LIN {X 0,Y 476.078,Z 721.43,A -85,B 0,C 180,E1 21900.686,E2 21900.686} C_VEL
LIN {X 0,Y 474.014,Z 739.797,A -85,B 0,C 180,E1 21899.021,E2 21899.021} C_VEL
LIN {X 0,Y 472.024,Z 756.489,A -85,B 0,C 180,E1 21897.228,E2 21897.228} C_VEL
LIN {X 0,Y 470.405,Z 770.596,A -85,B 0,C 180,E1 21895.493,E2 21895.493} C_VEL
LIN {X 0,Y 468.622,Z 786.231,A -85,B 0,C 180,E1 21893.248,E2 21893.248} C_VEL
LIN {X 0,Y 467.305,Z 798.417,A -85,B 0,C 180,E1 21891.198,E2 21891.198} C_VEL
LIN {X 0,Y 466.282,Z 809.049,A -85,B 0,C 180,E1 21889.152,E2 21889.152} C_VEL
LIN {X 0,Y 465.286,Z 820.849,A -85,B 0,C 180,E1 21886.478,E2 21886.478} C_VEL
LIN {X 0,Y 464.694,Z 829.202,A -85,B 0,C 180,E1 21884.198,E2 21884.198} C_VEL
LIN {X 0,Y 464.302,Z 836.544,A -85,B 0,C 180,E1 21881.805,E2 21881.805} C_VEL
LIN {X 0,Y 464.048,Z 843.148,A -85,B 0,C 180,E1 21879.049,E2 21879.049} C_VEL
LIN {X 0,Y 463.95,Z 847.377,A -85,B 0,C 180,E1 21876.683,E2 21876.683} C_VEL
LIN {X 0,Y 463.916,Z 850.478,A -85,B 0,C 180,E1 21874.202,E2 21874.202} C_VEL
LIN {X 0,Y 463.901,Z 852.199,A -85,B 0,C 180,E1 21871.482,E2 21871.482} C_VEL
LIN {X 0,Y 463.906,Z 852.333,A -85,B 0,C 180,E1 21869.136,E2 21869.136} C_VEL
LIN {X 0,Y 463.915,Z 851.272,A -85,B 0,C 180,E1 21866.788,E2 21866.788} C_VEL
LIN {X 0,Y 463.938,Z 848.514,A -85,B 0,C 180,E1 21864.062,E2 21864.062} C_VEL
LIN {X 0,Y 464.017,Z 844.133,A -85,B 0,C 180,E1 21861.45,E2 21861.45} C_VEL
LIN {X 0,Y 464.188,Z 839.084,A -85,B 0,C 180,E1 21859.179,E2 21859.179} C_VEL
LIN {X 0,Y 464.572,Z 831.33,A -85,B 0,C 180,E1 21856.433,E2 21856.433} C_VEL
LIN {X 0,Y 465.126,Z 822.811,A -85,B 0,C 180,E1 21854.029,E2 21854.029} C_VEL
LIN {X 0,Y 465.9,Z 813.253,A -85,B 0,C 180,E1 21851.741,E2 21851.741} C_VEL
LIN {X 0,Y 467.095,Z 800.545,A -85,B 0,C 180,E1 21849.186,E2 21849.186} C_VEL
LIN {X 0,Y 468.267,Z 789.404,A -85,B 0,C 180,E1 21847.265,E2 21847.265} C_VEL
LIN {X 0,Y 469.696,Z 776.705,A -85,B 0,C 180,E1 21845.341,E2 21845.341} C_VEL
LIN {X 0,Y 471.648,Z 759.814,A -85,B 0,C 180,E1 21843.158,E2 21843.158} C_VEL
LIN {X 0,Y 473.329,Z 745.351,A -85,B 0,C 180,E1 21841.554,E2 21841.554} C_VEL
LIN {X 0,Y 475.189,Z 729.447,A -85,B 0,C 180,E1 21840.009,E2 21840.009} C_VEL
LIN {X 0,Y 477.4,Z 709.425,A -85,B 0,C 180,E1 21838.357,E2 21838.357} C_VEL
LIN {X 0,Y 479.116,Z 692.979,A -85,B 0,C 180,E1 21837.212,E2 21837.212} C_VEL
LIN {X 0,Y 480.757,Z 675.933,A -85,B 0,C 180,E1 21836.198,E2 21836.198} C_VEL
LIN {X 0,Y 482.578,Z 654.654,A -85,B 0,C 180,E1 21835.158,E2 21835.158} C_VEL
LIN {X 0,Y 483.957,Z 634.596,A -85,B 0,C 180,E1 21834.403,E2 21834.403} C_VEL
LIN {X 0,Y 485.007,Z 616.285,A -85,B 0,C 180,E1 21833.877,E2 21833.877} C_VEL
LIN {X 0,Y 485.886,Z 591.815,A -85,B 0,C 180,E1 21833.389,E2 21833.389} C_VEL
LIN {X 0,Y 490.39,Z 370.649,A -85,B 0,C 180,E1 21829.748,E2 21829.748} C_VEL
LIN {X 0,Y 490.854,Z 340.827,A -85,B 0,C 180,E1 21829.233,E2 21829.233} C_VEL
LIN {X 0,Y 487.266,Z 328.463,A -85,B 0,C 180,E1 21828.634,E2 21828.634} C_VEL
LIN {X 0,Y 474.742,Z 306.974,A -85,B 0,C 180,E1 21826.867,E2 21826.867} C_VEL
LIN {X 0,Y 471.808,Z 301.758,A -85,B 0,C 180,E1 21826.372,E2 21826.372} C_VEL
LIN {X 0,Y 467.061,Z 288.332,A -85,B 0,C 180,E1 21823.746,E2 21823.746} C_VEL
LIN {X 0,Y 464.967,Z 282.439,A -85,B 0,C 180,E1 21822.471,E2 21822.471} C_VEL
LIN {X 0,Y 464.991,Z 282.262,A -85,B 0,C 180,E1 21819.052,E2 21819.052} C_VEL
LIN {X 0,Y 464.994,Z 282.317,A -85,B 0,C 180,E1 21815.42,E2 21815.42} C_VEL
LIN {X 0,Y 464.961,Z 282.319,A -85,B 0,C 180,E1 21811.855,E2 21811.855} C_VEL
LIN {X 0,Y 464.957,Z 282.317,A -85,B 0,C 180,E1 21808.235,E2 21808.235} C_VEL
LIN {X 0,Y 464.982,Z 282.302,A -85,B 0,C 180,E1 21804.655,E2 21804.655} C_VEL
LIN {X 0,Y 465.012,Z 282.287,A -85,B 0,C 180,E1 21801.068,E2 21801.068} C_VEL
LIN {X 0,Y 464.975,Z 282.314,A -85,B 0,C 180,E1 21797.521,E2 21797.521} C_VEL
LIN {X 0,Y 464.96,Z 282.299,A -85,B 0,C 180,E1 21793.936,E2 21793.936} C_VEL
LIN {X 0,Y 464.984,Z 282.3,A -85,B 0,C 180,E1 21790.406,E2 21790.406} C_VEL
LIN {X 0,Y 465.019,Z 282.307,A -85,B 0,C 180,E1 21786.792,E2 21786.792} C_VEL
LIN {X 0,Y 464.995,Z 282.287,A -85,B 0,C 180,E1 21783.081,E2 21783.081} C_VEL
LIN {X 0,Y 464.972,Z 282.315,A -85,B 0,C 180,E1 21779.507,E2 21779.507} C_VEL
LIN {X 0,Y 464.971,Z 282.294,A -85,B 0,C 180,E1 21775.807,E2 21775.807} C_VEL
LIN {X 0,Y 464.998,Z 282.304,A -85,B 0,C 180,E1 21772.215,E2 21772.215} C_VEL
LIN {X 0,Y 465.014,Z 282.303,A -85,B 0,C 180,E1 21768.591,E2 21768.591} C_VEL
LIN {X 0,Y 464.998,Z 282.289,A -85,B 0,C 180,E1 21764.919,E2 21764.919} C_VEL
LIN {X 0,Y 464.98,Z 282.315,A -85,B 0,C 180,E1 21761.313,E2 21761.313} C_VEL
LIN {X 0,Y 464.983,Z 282.313,A -85,B 0,C 180,E1 21757.609,E2 21757.609} C_VEL
LIN {X 0,Y 465.005,Z 282.311,A -85,B 0,C 180,E1 21753.983,E2 21753.983} C_VEL
LIN {X 0,Y 465.019,Z 282.311,A -85,B 0,C 180,E1 21750.3,E2 21750.3} C_VEL
LIN {X 0,Y 465.01,Z 282.311,A -85,B 0,C 180,E1 21746.602,E2 21746.602} C_VEL
LIN {X 0,Y 464.993,Z 282.314,A -85,B 0,C 180,E1 21742.913,E2 21742.913} C_VEL
LIN {X 0,Y 464.99,Z 282.313,A -85,B 0,C 180,E1 21739.343,E2 21739.343} C_VEL
LIN {X 0,Y 465.007,Z 282.311,A -85,B 0,C 180,E1 21735.668,E2 21735.668} C_VEL
LIN {X 0,Y 465.015,Z 282.312,A -85,B 0,C 180,E1 21731.931,E2 21731.931} C_VEL
LIN {X 0,Y 465.018,Z 282.312,A -85,B 0,C 180,E1 21728.26,E2 21728.26} C_VEL
LIN {X 0,Y 465.002,Z 282.312,A -85,B 0,C 180,E1 21724.56,E2 21724.56} C_VEL
LIN {X 0,Y 464.994,Z 282.311,A -85,B 0,C 180,E1 21720.913,E2 21720.913} C_VEL
LIN {X 0,Y 465.005,Z 282.307,A -85,B 0,C 180,E1 21717.257,E2 21717.257} C_VEL
LIN {X 0,Y 465.013,Z 282.308,A -85,B 0,C 180,E1 21713.573,E2 21713.573} C_VEL
LIN {X 0,Y 465.01,Z 282.31,A -85,B 0,C 180,E1 21709.86,E2 21709.86} C_VEL
LIN {X 0,Y 465.011,Z 282.31,A -85,B 0,C 180,E1 21709.539,E2 21709.539} C_VEL
LIN {X 0,Y 464.032,Z 282.435,A -85,B 0,C 180,E1 21708.59,E2 21708.59} C_VEL
LIN {X 0,Y 457.52,Z 283.245,A -85,B 0,C 180,E1 21705.85,E2 21705.85} C_VEL
LIN {X 0,Y 457.076,Z 283.3,A -85,B 0,C 180,E1 21705.223,E2 21705.223} C_VEL
LIN {X 0,Y 457.07,Z 283.302,A -85,B 0,C 180,E1 21701.474,E2 21701.474} C_VEL
LIN {X 0,Y 457.067,Z 283.304,A -85,B 0,C 180,E1 21697.71,E2 21697.71} C_VEL
LIN {X 0,Y 457.069,Z 283.302,A -85,B 0,C 180,E1 21694.014,E2 21694.014} C_VEL
LIN {X 0,Y 457.069,Z 283.301,A -85,B 0,C 180,E1 21690.251,E2 21690.251} C_VEL
LIN {X 0,Y 457.065,Z 283.301,A -85,B 0,C 180,E1 21686.488,E2 21686.488} C_VEL
LIN {X 0,Y 457.072,Z 283.3,A -85,B 0,C 180,E1 21682.711,E2 21682.711} C_VEL
LIN {X 0,Y 457.067,Z 283.301,A -85,B 0,C 180,E1 21679.029,E2 21679.029} C_VEL
LIN {X 0,Y 457.059,Z 283.304,A -85,B 0,C 180,E1 21675.3,E2 21675.3} C_VEL
LIN {X 0,Y 457.068,Z 283.302,A -85,B 0,C 180,E1 21671.639,E2 21671.639} C_VEL
LIN {X 0,Y 457.078,Z 283.299,A -85,B 0,C 180,E1 21667.899,E2 21667.899} C_VEL
LIN {X 0,Y 457.073,Z 283.298,A -85,B 0,C 180,E1 21664.195,E2 21664.195} C_VEL
LIN {X 0,Y 457.077,Z 283.297,A -85,B 0,C 180,E1 21660.516,E2 21660.516} C_VEL
LIN {X 0,Y 457.059,Z 283.3,A -85,B 0,C 180,E1 21656.847,E2 21656.847} C_VEL
LIN {X 0,Y 457.056,Z 283.301,A -85,B 0,C 180,E1 21653.174,E2 21653.174} C_VEL
LIN {X 0,Y 457.07,Z 283.3,A -85,B 0,C 180,E1 21649.483,E2 21649.483} C_VEL
LIN {X 0,Y 457.074,Z 283.3,A -85,B 0,C 180,E1 21645.749,E2 21645.749} C_VEL
LIN {X 0,Y 457.075,Z 283.301,A -85,B 0,C 180,E1 21642.019,E2 21642.019} C_VEL
LIN {X 0,Y 457.058,Z 283.301,A -85,B 0,C 180,E1 21638.409,E2 21638.409} C_VEL
LIN {X 0,Y 457.047,Z 283.304,A -85,B 0,C 180,E1 21634.818,E2 21634.818} C_VEL
LIN {X 0,Y 457.056,Z 283.303,A -85,B 0,C 180,E1 21631.083,E2 21631.083} C_VEL
LIN {X 0,Y 457.076,Z 283.302,A -85,B 0,C 180,E1 21627.488,E2 21627.488} C_VEL
LIN {X 0,Y 457.077,Z 283.3,A -85,B 0,C 180,E1 21623.735,E2 21623.735} C_VEL
LIN {X 0,Y 457.056,Z 283.3,A -85,B 0,C 180,E1 21620.087,E2 21620.087} C_VEL
LIN {X 0,Y 457.035,Z 283.286,A -85,B 0,C 180,E1 21616.523,E2 21616.523} C_VEL
LIN {X 0,Y 457.05,Z 283.305,A -85,B 0,C 180,E1 21612.893,E2 21612.893} C_VEL
LIN {X 0,Y 457.069,Z 283.273,A -85,B 0,C 180,E1 21609.189,E2 21609.189} C_VEL
LIN {X 0,Y 457.073,Z 283.296,A -85,B 0,C 180,E1 21605.523,E2 21605.523} C_VEL
LIN {X 0,Y 457.043,Z 283.292,A -85,B 0,C 180,E1 21601.88,E2 21601.88} C_VEL
LIN {X 0,Y 457.028,Z 283.286,A -85,B 0,C 180,E1 21598.245,E2 21598.245} C_VEL
LIN {X 0,Y 457.039,Z 283.305,A -85,B 0,C 180,E1 21594.602,E2 21594.602} C_VEL
LIN {X 0,Y 457.07,Z 283.272,A -85,B 0,C 180,E1 21591.065,E2 21591.065} C_VEL
LIN {X 0,Y 457.065,Z 283.301,A -85,B 0,C 180,E1 21587.324,E2 21587.324} C_VEL
LIN {X 0,Y 457.031,Z 283.294,A -85,B 0,C 180,E1 21583.738,E2 21583.738} C_VEL
LIN {X 0,Y 457.019,Z 283.283,A -85,B 0,C 180,E1 21580.044,E2 21580.044} C_VEL
LIN {X 0,Y 457.033,Z 283.303,A -85,B 0,C 180,E1 21576.4,E2 21576.4} C_VEL
LIN {X 0,Y 457.066,Z 283.291,A -85,B 0,C 180,E1 21572.794,E2 21572.794} C_VEL
LIN {X 0,Y 457.044,Z 283.29,A -85,B 0,C 180,E1 21569.209,E2 21569.209} C_VEL
LIN {X 0,Y 457.015,Z 283.297,A -85,B 0,C 180,E1 21565.636,E2 21565.636} C_VEL
LIN {X 0,Y 457.008,Z 283.254,A -85,B 0,C 180,E1 21561.905,E2 21561.905} C_VEL
LIN {X 0,Y 457.06,Z 283.456,A -85,B 0,C 180,E1 21558.358,E2 21558.358} C_VEL
LIN {X 0,Y 461.683,Z 296.244,A -85,B 0,C 180,E1 21555.612,E2 21555.612} C_VEL
LIN {X 0,Y 463.685,Z 301.866,A -85,B 0,C 180,E1 21554.548,E2 21554.548} C_VEL
LIN {X 0,Y 475.763,Z 322.216,A -85,B 0,C 180,E1 21552.713,E2 21552.713} C_VEL
LIN {X 0,Y 482.346,Z 334.147,A -85,B 0,C 180,E1 21551.767,E2 21551.767} C_VEL
LIN {X 0,Y 484.884,Z 344.128,A -85,B 0,C 180,E1 21551.31,E2 21551.31} C_VEL
LIN {X 0,Y 480.16,Z 557.469,A -85,B 0,C 180,E1 21547.748,E2 21547.748} C_VEL
LIN {X 0,Y 478.932,Z 607.783,A -85,B 0,C 180,E1 21546.884,E2 21546.884} C_VEL
LIN {X 0,Y 477.681,Z 630.638,A -85,B 0,C 180,E1 21546.282,E2 21546.282} C_VEL
LIN {X 0,Y 476.431,Z 648.133,A -85,B 0,C 180,E1 21545.653,E2 21545.653} C_VEL
LIN {X 0,Y 474.914,Z 666.067,A -85,B 0,C 180,E1 21544.852,E2 21544.852} C_VEL
LIN {X 0,Y 472.913,Z 686.795,A -85,B 0,C 180,E1 21543.709,E2 21543.709} C_VEL
LIN {X 0,Y 470.923,Z 704.82,A -85,B 0,C 180,E1 21542.49,E2 21542.49} C_VEL
LIN {X 0,Y 469.027,Z 721.175,A -85,B 0,C 180,E1 21541.199,E2 21541.199} C_VEL
LIN {X 0,Y 466.801,Z 739.54,A -85,B 0,C 180,E1 21539.514,E2 21539.514} C_VEL
LIN {X 0,Y 464.684,Z 756.232,A -85,B 0,C 180,E1 21537.694,E2 21537.694} C_VEL
LIN {X 0,Y 462.929,Z 770.339,A -85,B 0,C 180,E1 21535.935,E2 21535.935} C_VEL
LIN {X 0,Y 461.037,Z 786.153,A -85,B 0,C 180,E1 21533.653,E2 21533.653} C_VEL
LIN {X 0,Y 459.705,Z 797.705,A -85,B 0,C 180,E1 21531.7,E2 21531.7} C_VEL
LIN {X 0,Y 458.564,Z 808.414,A -85,B 0,C 180,E1 21529.62,E2 21529.62} C_VEL
LIN {X 0,Y 457.504,Z 819.863,A -85,B 0,C 180,E1 21527.028,E2 21527.028} C_VEL
LIN {X 0,Y 456.801,Z 828.772,A -85,B 0,C 180,E1 21524.579,E2 21524.579} C_VEL
LIN {X 0,Y 456.374,Z 835.814,A -85,B 0,C 180,E1 21522.269,E2 21522.269} C_VEL
LIN {X 0,Y 456.09,Z 842.729,A -85,B 0,C 180,E1 21519.424,E2 21519.424} C_VEL
LIN {X 0,Y 455.967,Z 847.183,A -85,B 0,C 180,E1 21516.927,E2 21516.927} C_VEL
LIN {X 0,Y 455.921,Z 850.204,A -85,B 0,C 180,E1 21514.528,E2 21514.528} C_VEL
LIN {X 0,Y 455.9,Z 852.143,A -85,B 0,C 180,E1 21511.759,E2 21511.759} C_VEL
LIN {X 0,Y 455.902,Z 852.357,A -85,B 0,C 180,E1 21509.246,E2 21509.246} C_VEL
LIN {X 0,Y 455.914,Z 851.429,A -85,B 0,C 180,E1 21506.983,E2 21506.983} C_VEL
LIN {X 0,Y 455.935,Z 848.989,A -85,B 0,C 180,E1 21504.337,E2 21504.337} C_VEL
LIN {X 0,Y 456.023,Z 844.623,A -85,B 0,C 180,E1 21501.553,E2 21501.553} C_VEL
LIN {X 0,Y 456.192,Z 839.74,A -85,B 0,C 180,E1 21499.263,E2 21499.263} C_VEL
LIN {X 0,Y 456.52,Z 833.268,A -85,B 0,C 180,E1 21496.834,E2 21496.834} C_VEL
LIN {X 0,Y 457.134,Z 824.278,A -85,B 0,C 180,E1 21494.134,E2 21494.134} C_VEL
LIN {X 0,Y 457.877,Z 815.484,A -85,B 0,C 180,E1 21491.936,E2 21491.936} C_VEL
LIN {X 0,Y 458.895,Z 805.256,A -85,B 0,C 180,E1 21489.731,E2 21489.731} C_VEL
LIN {X 0,Y 460.39,Z 791.775,A -85,B 0,C 180,E1 21487.259,E2 21487.259} C_VEL
LIN {X 0,Y 461.844,Z 779.199,A -85,B 0,C 180,E1 21485.303,E2 21485.303} C_VEL
LIN {X 0,Y 463.558,Z 765.359,A -85,B 0,C 180,E1 21483.413,E2 21483.413} C_VEL
LIN {X 0,Y 465.771,Z 747.562,A -85,B 0,C 180,E1 21481.33,E2 21481.33} C_VEL
LIN {X 0,Y 467.714,Z 731.973,A -85,B 0,C 180,E1 21479.766,E2 21479.766} C_VEL
LIN {X 0,Y 469.773,Z 714.998,A -85,B 0,C 180,E1 21478.285,E2 21478.285} C_VEL
LIN {X 0,Y 472.021,Z 695.017,A -85,B 0,C 180,E1 21476.824,E2 21476.824} C_VEL
LIN {X 0,Y 473.784,Z 677.949,A -85,B 0,C 180,E1 21475.778,E2 21475.778} C_VEL
LIN {X 0,Y 475.474,Z 659.965,A -85,B 0,C 180,E1 21474.855,E2 21474.855} C_VEL
LIN {X 0,Y 477.25,Z 636.858,A -85,B 0,C 180,E1 21473.922,E2 21473.922} C_VEL
LIN {X 0,Y 478.405,Z 618.224,A -85,B 0,C 180,E1 21473.365,E2 21473.365} C_VEL
LIN {X 0,Y 479.277,Z 598.293,A -85,B 0,C 180,E1 21472.935,E2 21472.935} C_VEL
LIN {X 0,Y 484.124,Z 377.411,A -85,B 0,C 180,E1 21469.251,E2 21469.251} C_VEL
LIN {X 0,Y 484.736,Z 342.818,A -85,B 0,C 180,E1 21468.65,E2 21468.65} C_VEL
LIN {X 0,Y 481.761,Z 332.731,A -85,B 0,C 180,E1 21468.143,E2 21468.143} C_VEL
LIN {X 0,Y 469.816,Z 312.108,A -85,B 0,C 180,E1 21466.411,E2 21466.411} C_VEL
LIN {X 0,Y 463.47,Z 301.409,A -85,B 0,C 180,E1 21465.391,E2 21465.391} C_VEL
LIN {X 0,Y 458.235,Z 286.749,A -85,B 0,C 180,E1 21462.394,E2 21462.394} C_VEL
LIN {X 0,Y 457.055,Z 283.397,A -85,B 0,C 180,E1 21461.601,E2 21461.601} C_VEL
LIN {X 0,Y 457.01,Z 283.254,A -85,B 0,C 180,E1 21458.039,E2 21458.039} C_VEL
LIN {X 0,Y 457.015,Z 283.297,A -85,B 0,C 180,E1 21454.364,E2 21454.364} C_VEL
LIN {X 0,Y 457.044,Z 283.29,A -85,B 0,C 180,E1 21450.791,E2 21450.791} C_VEL
LIN {X 0,Y 457.066,Z 283.291,A -85,B 0,C 180,E1 21447.206,E2 21447.206} C_VEL
LIN {X 0,Y 457.036,Z 283.302,A -85,B 0,C 180,E1 21443.563,E2 21443.563} C_VEL
LIN {X 0,Y 457.018,Z 283.281,A -85,B 0,C 180,E1 21439.956,E2 21439.956} C_VEL
LIN {X 0,Y 457.029,Z 283.291,A -85,B 0,C 180,E1 21436.262,E2 21436.262} C_VEL
LIN {X 0,Y 457.066,Z 283.299,A -85,B 0,C 180,E1 21432.677,E2 21432.677} C_VEL
LIN {X 0,Y 457.07,Z 283.272,A -85,B 0,C 180,E1 21428.935,E2 21428.935} C_VEL
LIN {X 0,Y 457.039,Z 283.306,A -85,B 0,C 180,E1 21425.398,E2 21425.398} C_VEL
LIN {X 0,Y 457.028,Z 283.286,A -85,B 0,C 180,E1 21421.755,E2 21421.755} C_VEL
LIN {X 0,Y 457.043,Z 283.292,A -85,B 0,C 180,E1 21418.12,E2 21418.12} C_VEL
LIN {X 0,Y 457.071,Z 283.297,A -85,B 0,C 180,E1 21414.442,E2 21414.442} C_VEL
LIN {X 0,Y 457.069,Z 283.273,A -85,B 0,C 180,E1 21410.811,E2 21410.811} C_VEL
LIN {X 0,Y 457.05,Z 283.305,A -85,B 0,C 180,E1 21407.107,E2 21407.107} C_VEL
LIN {X 0,Y 457.036,Z 283.286,A -85,B 0,C 180,E1 21403.477,E2 21403.477} C_VEL
LIN {X 0,Y 457.049,Z 283.3,A -85,B 0,C 180,E1 21399.779,E2 21399.779} C_VEL
LIN {X 0,Y 457.072,Z 283.3,A -85,B 0,C 180,E1 21396.115,E2 21396.115} C_VEL
LIN {X 0,Y 457.079,Z 283.301,A -85,B 0,C 180,E1 21392.364,E2 21392.364} C_VEL
LIN {X 0,Y 457.072,Z 283.3,A -85,B 0,C 180,E1 21388.625,E2 21388.625} C_VEL
LIN {X 0,Y 457.05,Z 283.304,A -85,B 0,C 180,E1 21385.029,E2 21385.029} C_VEL
LIN {X 0,Y 457.048,Z 283.303,A -85,B 0,C 180,E1 21381.269,E2 21381.269} C_VEL
LIN {X 0,Y 457.066,Z 283.3,A -85,B 0,C 180,E1 21377.642,E2 21377.642} C_VEL
LIN {X 0,Y 457.076,Z 283.301,A -85,B 0,C 180,E1 21373.902,E2 21373.902} C_VEL
LIN {X 0,Y 457.076,Z 283.301,A -85,B 0,C 180,E1 21370.188,E2 21370.188} C_VEL
LIN {X 0,Y 457.066,Z 283.3,A -85,B 0,C 180,E1 21366.513,E2 21366.513} C_VEL
LIN {X 0,Y 457.056,Z 283.3,A -85,B 0,C 180,E1 21362.855,E2 21362.855} C_VEL
LIN {X 0,Y 457.064,Z 283.298,A -85,B 0,C 180,E1 21359.197,E2 21359.197} C_VEL
LIN {X 0,Y 457.072,Z 283.296,A -85,B 0,C 180,E1 21355.527,E2 21355.527} C_VEL
LIN {X 0,Y 457.07,Z 283.298,A -85,B 0,C 180,E1 21351.831,E2 21351.831} C_VEL
LIN {X 0,Y 457.073,Z 283.299,A -85,B 0,C 180,E1 21348.097,E2 21348.097} C_VEL
LIN {X 0,Y 457.076,Z 283.3,A -85,B 0,C 180,E1 21345.223,E2 21345.223} C_VEL
LIN {X 0,Y 456.081,Z 283.425,A -85,B 0,C 180,E1 21344.257,E2 21344.257} C_VEL
LIN {X 0,Y 449.567,Z 284.237,A -85,B 0,C 180,E1 21341.47,E2 21341.47} C_VEL
LIN {X 0,Y 449.125,Z 284.291,A -85,B 0,C 180,E1 21340.831,E2 21340.831} C_VEL
LIN {X 0,Y 449.139,Z 284.288,A -85,B 0,C 180,E1 21337.033,E2 21337.033} C_VEL
LIN {X 0,Y 449.128,Z 284.288,A -85,B 0,C 180,E1 21333.318,E2 21333.318} C_VEL
LIN {X 0,Y 449.126,Z 284.289,A -85,B 0,C 180,E1 21329.617,E2 21329.617} C_VEL
LIN {X 0,Y 449.129,Z 284.289,A -85,B 0,C 180,E1 21325.821,E2 21325.821} C_VEL
LIN {X 0,Y 449.134,Z 284.289,A -85,B 0,C 180,E1 21322.067,E2 21322.067} C_VEL
LIN {X 0,Y 449.13,Z 284.29,A -85,B 0,C 180,E1 21318.312,E2 21318.312} C_VEL
LIN {X 0,Y 449.135,Z 284.289,A -85,B 0,C 180,E1 21314.506,E2 21314.506} C_VEL
LIN {X 0,Y 449.133,Z 284.288,A -85,B 0,C 180,E1 21310.718,E2 21310.718} C_VEL
LIN {X 0,Y 449.12,Z 284.289,A -85,B 0,C 180,E1 21307.071,E2 21307.071} C_VEL
LIN {X 0,Y 449.12,Z 284.289,A -85,B 0,C 180,E1 21303.276,E2 21303.276} C_VEL
LIN {X 0,Y 449.13,Z 284.289,A -85,B 0,C 180,E1 21299.498,E2 21299.498} C_VEL
LIN {X 0,Y 449.133,Z 284.29,A -85,B 0,C 180,E1 21295.681,E2 21295.681} C_VEL
LIN {X 0,Y 449.137,Z 284.291,A -85,B 0,C 180,E1 21291.929,E2 21291.929} C_VEL
LIN {X 0,Y 449.139,Z 284.289,A -85,B 0,C 180,E1 21288.225,E2 21288.225} C_VEL
LIN {X 0,Y 449.12,Z 284.29,A -85,B 0,C 180,E1 21284.529,E2 21284.529} C_VEL
LIN {X 0,Y 449.112,Z 284.292,A -85,B 0,C 180,E1 21280.806,E2 21280.806} C_VEL
LIN {X 0,Y 449.117,Z 284.291,A -85,B 0,C 180,E1 21277.108,E2 21277.108} C_VEL
LIN {X 0,Y 449.129,Z 284.289,A -85,B 0,C 180,E1 21273.358,E2 21273.358} C_VEL
LIN {X 0,Y 449.14,Z 284.288,A -85,B 0,C 180,E1 21269.617,E2 21269.617} C_VEL
LIN {X 0,Y 449.133,Z 284.289,A -85,B 0,C 180,E1 21265.87,E2 21265.87} C_VEL
LIN {X 0,Y 449.115,Z 284.291,A -85,B 0,C 180,E1 21262.164,E2 21262.164} C_VEL
LIN {X 0,Y 449.103,Z 284.292,A -85,B 0,C 180,E1 21258.43,E2 21258.43} C_VEL
LIN {X 0,Y 449.1,Z 284.27,A -85,B 0,C 180,E1 21254.703,E2 21254.703} C_VEL
LIN {X 0,Y 449.119,Z 284.274,A -85,B 0,C 180,E1 21251.038,E2 21251.038} C_VEL
LIN {X 0,Y 449.144,Z 284.283,A -85,B 0,C 180,E1 21247.29,E2 21247.29} C_VEL
LIN {X 0,Y 449.125,Z 284.259,A -85,B 0,C 180,E1 21243.574,E2 21243.574} C_VEL
LIN {X 0,Y 449.098,Z 284.291,A -85,B 0,C 180,E1 21240,E2 21240} C_VEL
LIN {X 0,Y 449.089,Z 284.271,A -85,B 0,C 180,E1 21236.298,E2 21236.298} C_VEL
LIN {X 0,Y 449.099,Z 284.279,A -85,B 0,C 180,E1 21232.581,E2 21232.581} C_VEL
LIN {X 0,Y 449.127,Z 284.283,A -85,B 0,C 180,E1 21228.962,E2 21228.962} C_VEL
LIN {X 0,Y 449.136,Z 284.26,A -85,B 0,C 180,E1 21225.167,E2 21225.167} C_VEL
LIN {X 0,Y 449.109,Z 284.29,A -85,B 0,C 180,E1 21221.436,E2 21221.436} C_VEL
LIN {X 0,Y 449.082,Z 284.289,A -85,B 0,C 180,E1 21217.846,E2 21217.846} C_VEL
LIN {X 0,Y 449.081,Z 284.27,A -85,B 0,C 180,E1 21214.088,E2 21214.088} C_VEL
LIN {X 0,Y 449.105,Z 284.279,A -85,B 0,C 180,E1 21210.514,E2 21210.514} C_VEL
LIN {X 0,Y 449.126,Z 284.279,A -85,B 0,C 180,E1 21206.829,E2 21206.829} C_VEL
LIN {X 0,Y 449.094,Z 284.262,A -85,B 0,C 180,E1 21203.209,E2 21203.209} C_VEL
LIN {X 0,Y 449.07,Z 284.265,A -85,B 0,C 180,E1 21199.616,E2 21199.616} C_VEL
LIN {X 0,Y 449.146,Z 284.644,A -85,B 0,C 180,E1 21199.188,E2 21199.188} C_VEL
LIN {X 0,Y 453.993,Z 297.997,A -85,B 0,C 180,E1 21196.248,E2 21196.248} C_VEL
LIN {X 0,Y 455.251,Z 301.253,A -85,B 0,C 180,E1 21195.612,E2 21195.612} C_VEL
LIN {X 0,Y 466.57,Z 319.99,A -85,B 0,C 180,E1 21193.802,E2 21193.802} C_VEL
LIN {X 0,Y 476.881,Z 338.287,A -85,B 0,C 180,E1 21192.27,E2 21192.27} C_VEL
LIN {X 0,Y 478.819,Z 346.044,A -85,B 0,C 180,E1 21191.908,E2 21191.908} C_VEL
LIN {X 0,Y 473.77,Z 559.959,A -85,B 0,C 180,E1 21188.297,E2 21188.297} C_VEL
LIN {X 0,Y 472.516,Z 607.847,A -85,B 0,C 180,E1 21187.463,E2 21187.463} C_VEL
LIN {X 0,Y 471.196,Z 630.494,A -85,B 0,C 180,E1 21186.858,E2 21186.858} C_VEL
LIN {X 0,Y 469.938,Z 647.185,A -85,B 0,C 180,E1 21186.257,E2 21186.257} C_VEL
LIN {X 0,Y 468.421,Z 664.334,A -85,B 0,C 180,E1 21185.491,E2 21185.491} C_VEL
LIN {X 0,Y 466.492,Z 683.366,A -85,B 0,C 180,E1 21184.46,E2 21184.46} C_VEL
LIN {X 0,Y 464.122,Z 703.782,A -85,B 0,C 180,E1 21183.092,E2 21183.092} C_VEL
LIN {X 0,Y 462.206,Z 719.375,A -85,B 0,C 180,E1 21181.858,E2 21181.858} C_VEL
LIN {X 0,Y 460.092,Z 735.671,A -85,B 0,C 180,E1 21180.374,E2 21180.374} C_VEL
LIN {X 0,Y 457.602,Z 754.313,A -85,B 0,C 180,E1 21178.374,E2 21178.374} C_VEL
LIN {X 0,Y 455.68,Z 768.587,A -85,B 0,C 180,E1 21176.59,E2 21176.59} C_VEL
LIN {X 0,Y 453.783,Z 783.418,A -85,B 0,C 180,E1 21174.47,E2 21174.47} C_VEL
LIN {X 0,Y 452.024,Z 797.523,A -85,B 0,C 180,E1 21172.088,E2 21172.088} C_VEL
LIN {X 0,Y 450.808,Z 808.381,A -85,B 0,C 180,E1 21169.971,E2 21169.971} C_VEL
LIN {X 0,Y 449.722,Z 819.281,A -85,B 0,C 180,E1 21167.487,E2 21167.487} C_VEL
LIN {X 0,Y 448.892,Z 828.767,A -85,B 0,C 180,E1 21164.841,E2 21164.841} C_VEL
LIN {X 0,Y 448.424,Z 835.811,A -85,B 0,C 180,E1 21162.49,E2 21162.49} C_VEL
LIN {X 0,Y 448.106,Z 842.65,A -85,B 0,C 180,E1 21159.633,E2 21159.633} C_VEL
LIN {X 0,Y 447.976,Z 847.179,A -85,B 0,C 180,E1 21157.051,E2 21157.051} C_VEL
LIN {X 0,Y 447.922,Z 850.199,A -85,B 0,C 180,E1 21154.609,E2 21154.609} C_VEL
LIN {X 0,Y 447.901,Z 852.14,A -85,B 0,C 180,E1 21151.791,E2 21151.791} C_VEL
LIN {X 0,Y 447.903,Z 852.355,A -85,B 0,C 180,E1 21149.233,E2 21149.233} C_VEL
LIN {X 0,Y 447.914,Z 851.425,A -85,B 0,C 180,E1 21146.929,E2 21146.929} C_VEL
LIN {X 0,Y 447.935,Z 849.12,A -85,B 0,C 180,E1 21144.364,E2 21144.364} C_VEL
LIN {X 0,Y 448.028,Z 844.866,A -85,B 0,C 180,E1 21141.53,E2 21141.53} C_VEL
LIN {X 0,Y 448.208,Z 840.042,A -85,B 0,C 180,E1 21139.2,E2 21139.2} C_VEL
LIN {X 0,Y 448.534,Z 833.993,A -85,B 0,C 180,E1 21136.858,E2 21136.858} C_VEL
LIN {X 0,Y 449.191,Z 825.097,A -85,B 0,C 180,E1 21134.068,E2 21134.068} C_VEL
LIN {X 0,Y 450.01,Z 816.039,A -85,B 0,C 180,E1 21131.743,E2 21131.743} C_VEL
LIN {X 0,Y 450.943,Z 807.099,A -85,B 0,C 180,E1 21129.764,E2 21129.764} C_VEL
LIN {X 0,Y 452.384,Z 794.647,A -85,B 0,C 180,E1 21127.383,E2 21127.383} C_VEL
LIN {X 0,Y 454.11,Z 780.608,A -85,B 0,C 180,E1 21125.113,E2 21125.113} C_VEL
LIN {X 0,Y 455.815,Z 767.591,A -85,B 0,C 180,E1 21123.278,E2 21123.278} C_VEL
LIN {X 0,Y 457.989,Z 751.543,A -85,B 0,C 180,E1 21121.296,E2 21121.296} C_VEL
LIN {X 0,Y 460.33,Z 733.853,A -85,B 0,C 180,E1 21119.453,E2 21119.453} C_VEL
LIN {X 0,Y 462.302,Z 718.603,A -85,B 0,C 180,E1 21118.077,E2 21118.077} C_VEL
LIN {X 0,Y 464.461,Z 701.085,A -85,B 0,C 180,E1 21116.706,E2 21116.706} C_VEL
LIN {X 0,Y 466.801,Z 680.321,A -85,B 0,C 180,E1 21115.366,E2 21115.366} C_VEL
LIN {X 0,Y 468.547,Z 663.014,A -85,B 0,C 180,E1 21114.445,E2 21114.445} C_VEL
LIN {X 0,Y 470.115,Z 645.048,A -85,B 0,C 180,E1 21113.656,E2 21113.656} C_VEL
LIN {X 0,Y 471.758,Z 621.581,A -85,B 0,C 180,E1 21112.875,E2 21112.875} C_VEL
LIN {X 0,Y 472.726,Z 602.319,A -85,B 0,C 180,E1 21112.43,E2 21112.43} C_VEL
LIN {X 0,Y 477.8,Z 388.131,A -85,B 0,C 180,E1 21108.809,E2 21108.809} C_VEL
LIN {X 0,Y 478.673,Z 344.868,A -85,B 0,C 180,E1 21108.053,E2 21108.053} C_VEL
LIN {X 0,Y 476.295,Z 336.962,A -85,B 0,C 180,E1 21107.64,E2 21107.64} C_VEL
LIN {X 0,Y 464.727,Z 316.911,A -85,B 0,C 180,E1 21105.917,E2 21105.917} C_VEL
LIN {X 0,Y 455.249,Z 301.25,A -85,B 0,C 180,E1 21104.388,E2 21104.388} C_VEL
LIN {X 0,Y 451.106,Z 290.154,A -85,B 0,C 180,E1 21102.056,E2 21102.056} C_VEL
LIN {X 0,Y 449.1,Z 284.389,A -85,B 0,C 180,E1 21100.717,E2 21100.717} C_VEL
LIN {X 0,Y 449.122,Z 284.246,A -85,B 0,C 180,E1 21097.268,E2 21097.268} C_VEL
LIN {X 0,Y 449.096,Z 284.28,A -85,B 0,C 180,E1 21093.629,E2 21093.629} C_VEL
LIN {X 0,Y 449.079,Z 284.279,A -85,B 0,C 180,E1 21089.995,E2 21089.995} C_VEL
LIN {X 0,Y 449.079,Z 284.271,A -85,B 0,C 180,E1 21086.203,E2 21086.203} C_VEL
LIN {X 0,Y 449.106,Z 284.288,A -85,B 0,C 180,E1 21082.653,E2 21082.653} C_VEL
LIN {X 0,Y 449.131,Z 284.276,A -85,B 0,C 180,E1 21078.967,E2 21078.967} C_VEL
LIN {X 0,Y 449.115,Z 284.262,A -85,B 0,C 180,E1 21075.23,E2 21075.23} C_VEL
LIN {X 0,Y 449.094,Z 284.293,A -85,B 0,C 180,E1 21071.559,E2 21071.559} C_VEL
LIN {X 0,Y 449.088,Z 284.277,A -85,B 0,C 180,E1 21067.806,E2 21067.806} C_VEL
LIN {X 0,Y 449.095,Z 284.277,A -85,B 0,C 180,E1 21064.085,E2 21064.085} C_VEL
LIN {X 0,Y 449.121,Z 284.29,A -85,B 0,C 180,E1 21060.383,E2 21060.383} C_VEL
LIN {X 0,Y 449.13,Z 284.259,A -85,B 0,C 180,E1 21056.673,E2 21056.673} C_VEL
LIN {X 0,Y 449.125,Z 284.29,A -85,B 0,C 180,E1 21052.967,E2 21052.967} C_VEL
LIN {X 0,Y 449.098,Z 284.272,A -85,B 0,C 180,E1 21049.351,E2 21049.351} C_VEL
LIN {X 0,Y 449.098,Z 284.277,A -85,B 0,C 180,E1 21045.692,E2 21045.692} C_VEL
LIN {X 0,Y 449.119,Z 284.29,A -85,B 0,C 180,E1 21041.974,E2 21041.974} C_VEL
LIN {X 0,Y 449.142,Z 284.29,A -85,B 0,C 180,E1 21038.313,E2 21038.313} C_VEL
LIN {X 0,Y 449.135,Z 284.291,A -85,B 0,C 180,E1 21034.554,E2 21034.554} C_VEL
LIN {X 0,Y 449.123,Z 284.29,A -85,B 0,C 180,E1 21030.821,E2 21030.821} C_VEL
LIN {X 0,Y 449.11,Z 284.294,A -85,B 0,C 180,E1 21027.097,E2 21027.097} C_VEL
LIN {X 0,Y 449.11,Z 284.292,A -85,B 0,C 180,E1 21023.37,E2 21023.37} C_VEL
LIN {X 0,Y 449.126,Z 284.29,A -85,B 0,C 180,E1 21019.622,E2 21019.622} C_VEL
LIN {X 0,Y 449.136,Z 284.289,A -85,B 0,C 180,E1 21015.83,E2 21015.83} C_VEL
LIN {X 0,Y 449.136,Z 284.29,A -85,B 0,C 180,E1 21012.072,E2 21012.072} C_VEL
LIN {X 0,Y 449.138,Z 284.288,A -85,B 0,C 180,E1 21008.395,E2 21008.395} C_VEL
LIN {X 0,Y 449.124,Z 284.289,A -85,B 0,C 180,E1 21004.588,E2 21004.588} C_VEL
LIN {X 0,Y 449.117,Z 284.288,A -85,B 0,C 180,E1 21000.948,E2 21000.948} C_VEL
LIN {X 0,Y 449.13,Z 284.285,A -85,B 0,C 180,E1 20997.296,E2 20997.296} C_VEL
LIN {X 0,Y 449.136,Z 284.286,A -85,B 0,C 180,E1 20993.482,E2 20993.482} C_VEL
LIN {X 0,Y 449.133,Z 284.287,A -85,B 0,C 180,E1 20989.665,E2 20989.665} C_VEL
LIN {X 0,Y 449.133,Z 284.288,A -85,B 0,C 180,E1 20985.891,E2 20985.891} C_VEL
LIN {X 0,Y 449.129,Z 284.288,A -85,B 0,C 180,E1 20982.209,E2 20982.209} C_VEL
LIN {X 0,Y 449.125,Z 284.291,A -85,B 0,C 180,E1 20980.831,E2 20980.831} C_VEL
LIN {X 0,Y 448.125,Z 284.416,A -85,B 0,C 180,E1 20979.848,E2 20979.848} C_VEL
LIN {X 0,Y 441.612,Z 285.226,A -85,B 0,C 180,E1 20977.01,E2 20977.01} C_VEL
LIN {X 0,Y 441.189,Z 285.277,A -85,B 0,C 180,E1 20976.359,E2 20976.359} C_VEL
LIN {X 0,Y 441.186,Z 285.276,A -85,B 0,C 180,E1 20972.598,E2 20972.598} C_VEL
LIN {X 0,Y 441.195,Z 285.275,A -85,B 0,C 180,E1 20968.831,E2 20968.831} C_VEL
LIN {X 0,Y 441.193,Z 285.276,A -85,B 0,C 180,E1 20965.06,E2 20965.06} C_VEL
LIN {X 0,Y 441.187,Z 285.278,A -85,B 0,C 180,E1 20961.267,E2 20961.267} C_VEL
LIN {X 0,Y 441.184,Z 285.279,A -85,B 0,C 180,E1 20957.434,E2 20957.434} C_VEL
LIN {X 0,Y 441.191,Z 285.278,A -85,B 0,C 180,E1 20953.68,E2 20953.68} C_VEL
LIN {X 0,Y 441.194,Z 285.277,A -85,B 0,C 180,E1 20949.851,E2 20949.851} C_VEL
LIN {X 0,Y 441.195,Z 285.276,A -85,B 0,C 180,E1 20946.068,E2 20946.068} C_VEL
LIN {X 0,Y 441.196,Z 285.275,A -85,B 0,C 180,E1 20942.318,E2 20942.318} C_VEL
LIN {X 0,Y 441.193,Z 285.276,A -85,B 0,C 180,E1 20938.586,E2 20938.586} C_VEL
LIN {X 0,Y 441.179,Z 285.278,A -85,B 0,C 180,E1 20934.856,E2 20934.856} C_VEL
LIN {X 0,Y 441.176,Z 285.279,A -85,B 0,C 180,E1 20931.019,E2 20931.019} C_VEL
LIN {X 0,Y 441.181,Z 285.278,A -85,B 0,C 180,E1 20927.247,E2 20927.247} C_VEL
LIN {X 0,Y 441.192,Z 285.277,A -85,B 0,C 180,E1 20923.516,E2 20923.516} C_VEL
LIN {X 0,Y 441.2,Z 285.276,A -85,B 0,C 180,E1 20919.723,E2 20919.723} C_VEL
LIN {X 0,Y 441.198,Z 285.278,A -85,B 0,C 180,E1 20915.941,E2 20915.941} C_VEL
LIN {X 0,Y 441.186,Z 285.279,A -85,B 0,C 180,E1 20912.18,E2 20912.18} C_VEL
LIN {X 0,Y 441.168,Z 285.281,A -85,B 0,C 180,E1 20908.568,E2 20908.568} C_VEL
LIN {X 0,Y 441.168,Z 285.282,A -85,B 0,C 180,E1 20904.789,E2 20904.789} C_VEL
LIN {X 0,Y 441.184,Z 285.282,A -85,B 0,C 180,E1 20901.121,E2 20901.121} C_VEL
LIN {X 0,Y 441.197,Z 285.27,A -85,B 0,C 180,E1 20897.406,E2 20897.406} C_VEL
LIN {X 0,Y 441.2,Z 285.269,A -85,B 0,C 180,E1 20893.632,E2 20893.632} C_VEL
LIN {X 0,Y 441.171,Z 285.249,A -85,B 0,C 180,E1 20889.918,E2 20889.918} C_VEL
LIN {X 0,Y 441.157,Z 285.281,A -85,B 0,C 180,E1 20886.246,E2 20886.246} C_VEL
LIN {X 0,Y 441.154,Z 285.258,A -85,B 0,C 180,E1 20882.468,E2 20882.468} C_VEL
LIN {X 0,Y 441.174,Z 285.265,A -85,B 0,C 180,E1 20878.831,E2 20878.831} C_VEL
LIN {X 0,Y 441.19,Z 285.271,A -85,B 0,C 180,E1 20875.06,E2 20875.06} C_VEL
LIN {X 0,Y 441.184,Z 285.249,A -85,B 0,C 180,E1 20871.398,E2 20871.398} C_VEL
LIN {X 0,Y 441.161,Z 285.281,A -85,B 0,C 180,E1 20867.699,E2 20867.699} C_VEL
LIN {X 0,Y 441.144,Z 285.262,A -85,B 0,C 180,E1 20864.083,E2 20864.083} C_VEL
LIN {X 0,Y 441.153,Z 285.261,A -85,B 0,C 180,E1 20860.401,E2 20860.401} C_VEL
LIN {X 0,Y 441.186,Z 285.282,A -85,B 0,C 180,E1 20856.776,E2 20856.776} C_VEL
LIN {X 0,Y 441.191,Z 285.264,A -85,B 0,C 180,E1 20852.951,E2 20852.951} C_VEL
LIN {X 0,Y 441.157,Z 285.267,A -85,B 0,C 180,E1 20849.34,E2 20849.34} C_VEL
LIN {X 0,Y 441.138,Z 285.273,A -85,B 0,C 180,E1 20845.642,E2 20845.642} C_VEL
LIN {X 0,Y 441.129,Z 285.226,A -85,B 0,C 180,E1 20841.858,E2 20841.858} C_VEL
LIN {X 0,Y 441.184,Z 285.545,A -85,B 0,C 180,E1 20840.148,E2 20840.148} C_VEL
LIN {X 0,Y 446.167,Z 298.998,A -85,B 0,C 180,E1 20837.058,E2 20837.058} C_VEL
LIN {X 0,Y 447.156,Z 301.358,A -85,B 0,C 180,E1 20836.649,E2 20836.649} C_VEL
LIN {X 0,Y 459.112,Z 320.69,A -85,B 0,C 180,E1 20834.679,E2 20834.679} C_VEL
LIN {X 0,Y 471.266,Z 341.92,A -85,B 0,C 180,E1 20832.815,E2 20832.815} C_VEL
LIN {X 0,Y 472.8,Z 348.217,A -85,B 0,C 180,E1 20832.517,E2 20832.517} C_VEL
LIN {X 0,Y 467.437,Z 561.972,A -85,B 0,C 180,E1 20828.869,E2 20828.869} C_VEL
LIN {X 0,Y 466.152,Z 607.908,A -85,B 0,C 180,E1 20828.057,E2 20828.057} C_VEL
LIN {X 0,Y 464.763,Z 630.31,A -85,B 0,C 180,E1 20827.453,E2 20827.453} C_VEL
LIN {X 0,Y 463.375,Z 647.649,A -85,B 0,C 180,E1 20826.819,E2 20826.819} C_VEL
LIN {X 0,Y 461.707,Z 665.402,A -85,B 0,C 180,E1 20826.011,E2 20826.011} C_VEL
LIN {X 0,Y 459.423,Z 686.287,A -85,B 0,C 180,E1 20824.839,E2 20824.839} C_VEL
LIN {X 0,Y 457.106,Z 704.862,A -85,B 0,C 180,E1 20823.552,E2 20823.552} C_VEL
LIN {X 0,Y 454.938,Z 721.436,A -85,B 0,C 180,E1 20822.205,E2 20822.205} C_VEL
LIN {X 0,Y 452.214,Z 740.878,A -85,B 0,C 180,E1 20820.345,E2 20820.345} C_VEL
LIN {X 0,Y 450.073,Z 755.858,A -85,B 0,C 180,E1 20818.657,E2 20818.657} C_VEL
LIN {X 0,Y 448.074,Z 769.824,A -85,B 0,C 180,E1 20816.863,E2 20816.863} C_VEL
LIN {X 0,Y 445.817,Z 786.18,A -85,B 0,C 180,E1 20814.418,E2 20814.418} C_VEL
LIN {X 0,Y 444.242,Z 798.138,A -85,B 0,C 180,E1 20812.326,E2 20812.326} C_VEL
LIN {X 0,Y 442.919,Z 809.246,A -85,B 0,C 180,E1 20810.101,E2 20810.101} C_VEL
LIN {X 0,Y 441.709,Z 820.739,A -85,B 0,C 180,E1 20807.385,E2 20807.385} C_VEL
LIN {X 0,Y 440.992,Z 828.763,A -85,B 0,C 180,E1 20805.113,E2 20805.113} C_VEL
LIN {X 0,Y 440.501,Z 835.444,A -85,B 0,C 180,E1 20802.852,E2 20802.852} C_VEL
LIN {X 0,Y 440.144,Z 842.148,A -85,B 0,C 180,E1 20800.074,E2 20800.074} C_VEL
LIN {X 0,Y 439.983,Z 846.985,A -85,B 0,C 180,E1 20797.311,E2 20797.311} C_VEL
LIN {X 0,Y 439.927,Z 849.925,A -85,B 0,C 180,E1 20794.954,E2 20794.954} C_VEL
LIN {X 0,Y 439.909,Z 851.906,A -85,B 0,C 180,E1 20792.345,E2 20792.345} C_VEL
LIN {X 0,Y 439.899,Z 852.406,A -85,B 0,C 180,E1 20789.479,E2 20789.479} C_VEL
LIN {X 0,Y 439.914,Z 851.502,A -85,B 0,C 180,E1 20787.004,E2 20787.004} C_VEL
LIN {X 0,Y 439.935,Z 849.385,A -85,B 0,C 180,E1 20784.523,E2 20784.523} C_VEL
LIN {X 0,Y 440.032,Z 845.356,A -85,B 0,C 180,E1 20781.638,E2 20781.638} C_VEL
LIN {X 0,Y 440.223,Z 840.345,A -85,B 0,C 180,E1 20779.134,E2 20779.134} C_VEL
LIN {X 0,Y 440.56,Z 834.52,A -85,B 0,C 180,E1 20776.81,E2 20776.81} C_VEL
LIN {X 0,Y 441.181,Z 826.63,A -85,B 0,C 180,E1 20774.22,E2 20774.22} C_VEL
LIN {X 0,Y 442.131,Z 816.432,A -85,B 0,C 180,E1 20771.543,E2 20771.543} C_VEL
LIN {X 0,Y 443.189,Z 806.842,A -85,B 0,C 180,E1 20769.394,E2 20769.394} C_VEL
LIN {X 0,Y 444.642,Z 795.109,A -85,B 0,C 180,E1 20767.107,E2 20767.107} C_VEL
LIN {X 0,Y 446.582,Z 780.474,A -85,B 0,C 180,E1 20764.683,E2 20764.683} C_VEL
LIN {X 0,Y 448.429,Z 767.334,A -85,B 0,C 180,E1 20762.802,E2 20762.802} C_VEL
LIN {X 0,Y 450.662,Z 751.84,A -85,B 0,C 180,E1 20760.858,E2 20760.858} C_VEL
LIN {X 0,Y 453.154,Z 734.286,A -85,B 0,C 180,E1 20758.99,E2 20758.99} C_VEL
LIN {X 0,Y 455.342,Z 718.348,A -85,B 0,C 180,E1 20757.529,E2 20757.529} C_VEL
LIN {X 0,Y 457.752,Z 700.048,A -85,B 0,C 180,E1 20756.085,E2 20756.085} C_VEL
LIN {X 0,Y 460.119,Z 680.101,A -85,B 0,C 180,E1 20754.792,E2 20754.792} C_VEL
LIN {X 0,Y 461.969,Z 662.761,A -85,B 0,C 180,E1 20753.86,E2 20753.86} C_VEL
LIN {X 0,Y 463.649,Z 644.496,A -85,B 0,C 180,E1 20753.051,E2 20753.051} C_VEL
LIN {X 0,Y 465.379,Z 621.179,A -85,B 0,C 180,E1 20752.273,E2 20752.273} C_VEL
LIN {X 0,Y 466.386,Z 602.07,A -85,B 0,C 180,E1 20751.829,E2 20751.829} C_VEL
LIN {X 0,Y 471.784,Z 387.665,A -85,B 0,C 180,E1 20748.162,E2 20748.162} C_VEL
LIN {X 0,Y 472.663,Z 346.904,A -85,B 0,C 180,E1 20747.441,E2 20747.441} C_VEL
LIN {X 0,Y 470.869,Z 341.168,A -85,B 0,C 180,E1 20747.126,E2 20747.126} C_VEL
LIN {X 0,Y 457.72,Z 318.257,A -85,B 0,C 180,E1 20745.097,E2 20745.097} C_VEL
LIN {X 0,Y 448.854,Z 304.297,A -85,B 0,C 180,E1 20743.651,E2 20743.651} C_VEL
LIN {X 0,Y 446.57,Z 300.188,A -85,B 0,C 180,E1 20743.185,E2 20743.185} C_VEL
LIN {X 0,Y 442.071,Z 288.153,A -85,B 0,C 180,E1 20740.475,E2 20740.475} C_VEL
LIN {X 0,Y 441.162,Z 285.365,A -85,B 0,C 180,E1 20739.765,E2 20739.765} C_VEL
LIN {X 0,Y 441.136,Z 285.274,A -85,B 0,C 180,E1 20736.108,E2 20736.108} C_VEL
LIN {X 0,Y 441.14,Z 285.285,A -85,B 0,C 180,E1 20732.286,E2 20732.286} C_VEL
LIN {X 0,Y 441.167,Z 285.281,A -85,B 0,C 180,E1 20728.709,E2 20728.709} C_VEL
LIN {X 0,Y 441.187,Z 285.256,A -85,B 0,C 180,E1 20724.975,E2 20724.975} C_VEL
LIN {X 0,Y 441.178,Z 285.253,A -85,B 0,C 180,E1 20721.261,E2 20721.261} C_VEL
LIN {X 0,Y 441.151,Z 285.281,A -85,B 0,C 180,E1 20717.68,E2 20717.68} C_VEL
LIN {X 0,Y 441.145,Z 285.261,A -85,B 0,C 180,E1 20713.901,E2 20713.901} C_VEL
LIN {X 0,Y 441.154,Z 285.262,A -85,B 0,C 180,E1 20710.182,E2 20710.182} C_VEL
LIN {X 0,Y 441.183,Z 285.28,A -85,B 0,C 180,E1 20706.506,E2 20706.506} C_VEL
LIN {X 0,Y 441.192,Z 285.246,A -85,B 0,C 180,E1 20702.728,E2 20702.728} C_VEL
LIN {X 0,Y 441.189,Z 285.275,A -85,B 0,C 180,E1 20698.961,E2 20698.961} C_VEL
LIN {X 0,Y 441.168,Z 285.263,A -85,B 0,C 180,E1 20695.19,E2 20695.19} C_VEL
LIN {X 0,Y 441.156,Z 285.261,A -85,B 0,C 180,E1 20691.528,E2 20691.528} C_VEL
LIN {X 0,Y 441.159,Z 285.281,A -85,B 0,C 180,E1 20687.699,E2 20687.699} C_VEL
LIN {X 0,Y 441.18,Z 285.251,A -85,B 0,C 180,E1 20684.084,E2 20684.084} C_VEL
LIN {X 0,Y 441.2,Z 285.279,A -85,B 0,C 180,E1 20680.403,E2 20680.403} C_VEL
LIN {X 0,Y 441.198,Z 285.281,A -85,B 0,C 180,E1 20676.606,E2 20676.606} C_VEL
LIN {X 0,Y 441.181,Z 285.282,A -85,B 0,C 180,E1 20672.901,E2 20672.901} C_VEL
LIN {X 0,Y 441.169,Z 285.282,A -85,B 0,C 180,E1 20669.189,E2 20669.189} C_VEL
LIN {X 0,Y 441.17,Z 285.281,A -85,B 0,C 180,E1 20665.353,E2 20665.353} C_VEL
LIN {X 0,Y 441.181,Z 285.28,A -85,B 0,C 180,E1 20661.613,E2 20661.613} C_VEL
LIN {X 0,Y 441.196,Z 285.279,A -85,B 0,C 180,E1 20657.871,E2 20657.871} C_VEL
LIN {X 0,Y 441.198,Z 285.278,A -85,B 0,C 180,E1 20654.078,E2 20654.078} C_VEL
LIN {X 0,Y 441.2,Z 285.278,A -85,B 0,C 180,E1 20650.23,E2 20650.23} C_VEL
LIN {X 0,Y 441.192,Z 285.278,A -85,B 0,C 180,E1 20646.423,E2 20646.423} C_VEL
LIN {X 0,Y 441.183,Z 285.278,A -85,B 0,C 180,E1 20642.641,E2 20642.641} C_VEL
LIN {X 0,Y 441.179,Z 285.277,A -85,B 0,C 180,E1 20638.863,E2 20638.863} C_VEL
LIN {X 0,Y 441.184,Z 285.276,A -85,B 0,C 180,E1 20635.074,E2 20635.074} C_VEL
LIN {X 0,Y 441.195,Z 285.276,A -85,B 0,C 180,E1 20631.259,E2 20631.259} C_VEL
LIN {X 0,Y 441.195,Z 285.277,A -85,B 0,C 180,E1 20627.406,E2 20627.406} C_VEL
LIN {X 0,Y 441.191,Z 285.278,A -85,B 0,C 180,E1 20623.632,E2 20623.632} C_VEL
LIN {X 0,Y 441.191,Z 285.279,A -85,B 0,C 180,E1 20619.786,E2 20619.786} C_VEL
LIN {X 0,Y 441.189,Z 285.277,A -85,B 0,C 180,E1 20616.359,E2 20616.359} C_VEL
LIN {X 0,Y 440.218,Z 285.403,A -85,B 0,C 180,E1 20615.359,E2 20615.359} C_VEL
LIN {X 0,Y 433.694,Z 286.221,A -85,B 0,C 180,E1 20612.469,E2 20612.469} C_VEL
LIN {X 0,Y 433.253,Z 286.269,A -85,B 0,C 180,E1 20611.807,E2 20611.807} C_VEL
LIN {X 0,Y 433.255,Z 286.269,A -85,B 0,C 180,E1 20608.016,E2 20608.016} C_VEL
LIN {X 0,Y 433.254,Z 286.269,A -85,B 0,C 180,E1 20604.172,E2 20604.172} C_VEL
LIN {X 0,Y 433.253,Z 286.268,A -85,B 0,C 180,E1 20600.301,E2 20600.301} C_VEL
LIN {X 0,Y 433.256,Z 286.267,A -85,B 0,C 180,E1 20596.522,E2 20596.522} C_VEL
LIN {X 0,Y 433.256,Z 286.266,A -85,B 0,C 180,E1 20592.681,E2 20592.681} C_VEL
LIN {X 0,Y 433.255,Z 286.265,A -85,B 0,C 180,E1 20588.803,E2 20588.803} C_VEL
LIN {X 0,Y 433.243,Z 286.266,A -85,B 0,C 180,E1 20585.019,E2 20585.019} C_VEL
LIN {X 0,Y 433.241,Z 286.266,A -85,B 0,C 180,E1 20581.162,E2 20581.162} C_VEL
LIN {X 0,Y 433.246,Z 286.266,A -85,B 0,C 180,E1 20577.39,E2 20577.39} C_VEL
LIN {X 0,Y 433.254,Z 286.266,A -85,B 0,C 180,E1 20573.624,E2 20573.624} C_VEL
LIN {X 0,Y 433.26,Z 286.266,A -85,B 0,C 180,E1 20569.806,E2 20569.806} C_VEL
LIN {X 0,Y 433.258,Z 286.268,A -85,B 0,C 180,E1 20566.003,E2 20566.003} C_VEL
LIN {X 0,Y 433.256,Z 286.268,A -85,B 0,C 180,E1 20562.188,E2 20562.188} C_VEL
LIN {X 0,Y 433.243,Z 286.269,A -85,B 0,C 180,E1 20558.375,E2 20558.375} C_VEL
LIN {X 0,Y 433.232,Z 286.27,A -85,B 0,C 180,E1 20554.593,E2 20554.593} C_VEL
LIN {X 0,Y 433.231,Z 286.272,A -85,B 0,C 180,E1 20550.821,E2 20550.821} C_VEL
LIN {X 0,Y 433.239,Z 286.27,A -85,B 0,C 180,E1 20547.025,E2 20547.025} C_VEL
LIN {X 0,Y 433.253,Z 286.27,A -85,B 0,C 180,E1 20543.243,E2 20543.243} C_VEL
LIN {X 0,Y 433.259,Z 286.269,A -85,B 0,C 180,E1 20539.409,E2 20539.409} C_VEL
LIN {X 0,Y 433.26,Z 286.234,A -85,B 0,C 180,E1 20535.527,E2 20535.527} C_VEL
LIN {X 0,Y 433.249,Z 286.263,A -85,B 0,C 180,E1 20531.718,E2 20531.718} C_VEL
LIN {X 0,Y 433.23,Z 286.258,A -85,B 0,C 180,E1 20527.96,E2 20527.96} C_VEL
LIN {X 0,Y 433.216,Z 286.243,A -85,B 0,C 180,E1 20524.235,E2 20524.235} C_VEL
LIN {X 0,Y 433.217,Z 286.271,A -85,B 0,C 180,E1 20520.397,E2 20520.397} C_VEL
LIN {X 0,Y 433.223,Z 286.239,A -85,B 0,C 180,E1 20516.692,E2 20516.692} C_VEL
LIN {X 0,Y 433.252,Z 286.257,A -85,B 0,C 180,E1 20512.974,E2 20512.974} C_VEL
LIN {X 0,Y 433.254,Z 286.257,A -85,B 0,C 180,E1 20509.092,E2 20509.092} C_VEL
LIN {X 0,Y 433.253,Z 286.236,A -85,B 0,C 180,E1 20505.226,E2 20505.226} C_VEL
LIN {X 0,Y 433.231,Z 286.266,A -85,B 0,C 180,E1 20501.428,E2 20501.428} C_VEL
LIN {X 0,Y 433.207,Z 286.266,A -85,B 0,C 180,E1 20497.743,E2 20497.743} C_VEL
LIN {X 0,Y 433.201,Z 286.246,A -85,B 0,C 180,E1 20493.99,E2 20493.99} C_VEL
LIN {X 0,Y 433.209,Z 286.255,A -85,B 0,C 180,E1 20490.25,E2 20490.25} C_VEL
LIN {X 0,Y 433.24,Z 286.255,A -85,B 0,C 180,E1 20486.66,E2 20486.66} C_VEL
LIN {X 0,Y 433.234,Z 286.225,A -85,B 0,C 180,E1 20482.961,E2 20482.961} C_VEL
LIN {X 0,Y 433.261,Z 286.527,A -85,B 0,C 180,E1 20481.139,E2 20481.139} C_VEL
LIN {X 0,Y 438.276,Z 299.88,A -85,B 0,C 180,E1 20477.966,E2 20477.966} C_VEL
LIN {X 0,Y 445.69,Z 311.685,A -85,B 0,C 180,E1 20476.604,E2 20476.604} C_VEL
LIN {X 0,Y 456.945,Z 330.302,A -85,B 0,C 180,E1 20474.739,E2 20474.739} C_VEL
LIN {X 0,Y 466.241,Z 347.196,A -85,B 0,C 180,E1 20473.276,E2 20473.276} C_VEL
LIN {X 0,Y 466.839,Z 350.334,A -85,B 0,C 180,E1 20473.143,E2 20473.143} C_VEL
LIN {X 0,Y 461.152,Z 563.962,A -85,B 0,C 180,E1 20469.457,E2 20469.457} C_VEL
LIN {X 0,Y 459.834,Z 608.086,A -85,B 0,C 180,E1 20468.666,E2 20468.666} C_VEL
LIN {X 0,Y 458.369,Z 630.292,A -85,B 0,C 180,E1 20468.058,E2 20468.058} C_VEL
LIN {X 0,Y 456.861,Z 648.1,A -85,B 0,C 180,E1 20467.398,E2 20467.398} C_VEL
LIN {X 0,Y 455.032,Z 666.47,A -85,B 0,C 180,E1 20466.545,E2 20466.545} C_VEL
LIN {X 0,Y 452.486,Z 688.01,A -85,B 0,C 180,E1 20465.297,E2 20465.297} C_VEL
LIN {X 0,Y 450.181,Z 705.478,A -85,B 0,C 180,E1 20464.062,E2 20464.062} C_VEL
LIN {X 0,Y 447.8,Z 722.648,A -85,B 0,C 180,E1 20462.638,E2 20462.638} C_VEL
LIN {X 0,Y 444.911,Z 741.856,A -85,B 0,C 180,E1 20460.747,E2 20460.747} C_VEL
LIN {X 0,Y 442.676,Z 756.569,A -85,B 0,C 180,E1 20459.052,E2 20459.052} C_VEL
LIN {X 0,Y 440.408,Z 771.559,A -85,B 0,C 180,E1 20457.077,E2 20457.077} C_VEL
LIN {X 0,Y 438.116,Z 786.987,A -85,B 0,C 180,E1 20454.685,E2 20454.685} C_VEL
LIN {X 0,Y 436.495,Z 798.55,A -85,B 0,C 180,E1 20452.612,E2 20452.612} C_VEL
LIN {X 0,Y 434.999,Z 810.43,A -85,B 0,C 180,E1 20450.168,E2 20450.168} C_VEL
LIN {X 0,Y 433.747,Z 821.48,A -85,B 0,C 180,E1 20447.437,E2 20447.437} C_VEL
LIN {X 0,Y 433.006,Z 829.407,A -85,B 0,C 180,E1 20445.125,E2 20445.125} C_VEL
LIN {X 0,Y 432.44,Z 837.188,A -85,B 0,C 180,E1 20442.417,E2 20442.417} C_VEL
LIN {X 0,Y 432.121,Z 843.174,A -85,B 0,C 180,E1 20439.704,E2 20439.704} C_VEL
LIN {X 0,Y 431.985,Z 847.171,A -85,B 0,C 180,E1 20437.313,E2 20437.313} C_VEL
LIN {X 0,Y 431.927,Z 850.056,A -85,B 0,C 180,E1 20434.913,E2 20434.913} C_VEL
LIN {X 0,Y 431.908,Z 852.057,A -85,B 0,C 180,E1 20432.123,E2 20432.123} C_VEL
LIN {X 0,Y 431.9,Z 852.377,A -85,B 0,C 180,E1 20429.337,E2 20429.337} C_VEL
LIN {X 0,Y 431.914,Z 851.499,A -85,B 0,C 180,E1 20426.948,E2 20426.948} C_VEL
LIN {X 0,Y 431.936,Z 849.447,A -85,B 0,C 180,E1 20424.486,E2 20424.486} C_VEL
LIN {X 0,Y 432.036,Z 845.599,A -85,B 0,C 180,E1 20421.617,E2 20421.617} C_VEL
LIN {X 0,Y 432.252,Z 840.331,A -85,B 0,C 180,E1 20418.931,E2 20418.931} C_VEL
LIN {X 0,Y 432.601,Z 834.599,A -85,B 0,C 180,E1 20416.637,E2 20416.637} C_VEL
LIN {X 0,Y 433.198,Z 827.243,A -85,B 0,C 180,E1 20414.196,E2 20414.196} C_VEL
LIN {X 0,Y 434.251,Z 816.744,A -85,B 0,C 180,E1 20411.335,E2 20411.335} C_VEL
LIN {X 0,Y 435.373,Z 807.226,A -85,B 0,C 180,E1 20409.148,E2 20409.148} C_VEL
LIN {X 0,Y 436.811,Z 796.257,A -85,B 0,C 180,E1 20406.952,E2 20406.952} C_VEL
LIN {X 0,Y 438.973,Z 781.112,A -85,B 0,C 180,E1 20404.357,E2 20404.357} C_VEL
LIN {X 0,Y 440.998,Z 767.575,A -85,B 0,C 180,E1 20402.378,E2 20402.378} C_VEL
LIN {X 0,Y 443.273,Z 752.691,A -85,B 0,C 180,E1 20400.473,E2 20400.473} C_VEL
LIN {X 0,Y 446.106,Z 734.029,A -85,B 0,C 180,E1 20398.444,E2 20398.444} C_VEL
LIN {X 0,Y 448.419,Z 718.141,A -85,B 0,C 180,E1 20396.969,E2 20396.969} C_VEL
LIN {X 0,Y 450.874,Z 700.577,A -85,B 0,C 180,E1 20395.565,E2 20395.565} C_VEL
LIN {X 0,Y 453.479,Z 679.931,A -85,B 0,C 180,E1 20394.203,E2 20394.203} C_VEL
LIN {X 0,Y 455.443,Z 662.457,A -85,B 0,C 180,E1 20393.255,E2 20393.255} C_VEL
LIN {X 0,Y 457.282,Z 643.461,A -85,B 0,C 180,E1 20392.409,E2 20392.409} C_VEL
LIN {X 0,Y 459.063,Z 620.624,A -85,B 0,C 180,E1 20391.651,E2 20391.651} C_VEL
LIN {X 0,Y 460.104,Z 601.612,A -85,B 0,C 180,E1 20391.206,E2 20391.206} C_VEL
LIN {X 0,Y 465.84,Z 386.868,A -85,B 0,C 180,E1 20387.493,E2 20387.493} C_VEL
LIN {X 0,Y 466.709,Z 348.97,A -85,B 0,C 180,E1 20386.814,E2 20386.814} C_VEL
LIN {X 0,Y 465.554,Z 345.605,A -85,B 0,C 180,E1 20386.612,E2 20386.612} C_VEL
LIN {X 0,Y 453.089,Z 323.677,A -85,B 0,C 180,E1 20384.634,E2 20384.634} C_VEL
LIN {X 0,Y 444.318,Z 309.712,A -85,B 0,C 180,E1 20383.165,E2 20383.165} C_VEL
LIN {X 0,Y 438.272,Z 299.875,A -85,B 0,C 180,E1 20382.034,E2 20382.034} C_VEL
LIN {X 0,Y 433.245,Z 286.441,A -85,B 0,C 180,E1 20378.827,E2 20378.827} C_VEL
LIN {X 0,Y 433.238,Z 286.272,A -85,B 0,C 180,E1 20375.399,E2 20375.399} C_VEL
LIN {X 0,Y 433.222,Z 286.269,A -85,B 0,C 180,E1 20371.595,E2 20371.595} C_VEL
LIN {X 0,Y 433.203,Z 286.275,A -85,B 0,C 180,E1 20367.939,E2 20367.939} C_VEL
LIN {X 0,Y 433.205,Z 286.266,A -85,B 0,C 180,E1 20364.112,E2 20364.112} C_VEL
LIN {X 0,Y 433.213,Z 286.239,A -85,B 0,C 180,E1 20360.396,E2 20360.396} C_VEL
LIN {X 0,Y 433.244,Z 286.256,A -85,B 0,C 180,E1 20356.719,E2 20356.719} C_VEL
LIN {X 0,Y 433.256,Z 286.257,A -85,B 0,C 180,E1 20352.935,E2 20352.935} C_VEL
LIN {X 0,Y 433.237,Z 286.236,A -85,B 0,C 180,E1 20349.163,E2 20349.163} C_VEL
LIN {X 0,Y 433.218,Z 286.272,A -85,B 0,C 180,E1 20345.563,E2 20345.563} C_VEL
LIN {X 0,Y 433.211,Z 286.248,A -85,B 0,C 180,E1 20341.719,E2 20341.719} C_VEL
LIN {X 0,Y 433.221,Z 286.254,A -85,B 0,C 180,E1 20338.016,E2 20338.016} C_VEL
LIN {X 0,Y 433.246,Z 286.265,A -85,B 0,C 180,E1 20334.305,E2 20334.305} C_VEL
LIN {X 0,Y 433.255,Z 286.233,A -85,B 0,C 180,E1 20330.569,E2 20330.569} C_VEL
LIN {X 0,Y 433.254,Z 286.264,A -85,B 0,C 180,E1 20326.793,E2 20326.793} C_VEL
LIN {X 0,Y 433.231,Z 286.253,A -85,B 0,C 180,E1 20323.094,E2 20323.094} C_VEL
LIN {X 0,Y 433.226,Z 286.27,A -85,B 0,C 180,E1 20319.322,E2 20319.322} C_VEL
LIN {X 0,Y 433.228,Z 286.27,A -85,B 0,C 180,E1 20315.454,E2 20315.454} C_VEL
LIN {X 0,Y 433.235,Z 286.27,A -85,B 0,C 180,E1 20311.613,E2 20311.613} C_VEL
LIN {X 0,Y 433.25,Z 286.268,A -85,B 0,C 180,E1 20307.881,E2 20307.881} C_VEL
LIN {X 0,Y 433.259,Z 286.266,A -85,B 0,C 180,E1 20304.096,E2 20304.096} C_VEL
LIN {X 0,Y 433.261,Z 286.265,A -85,B 0,C 180,E1 20300.216,E2 20300.216} C_VEL
LIN {X 0,Y 433.256,Z 286.265,A -85,B 0,C 180,E1 20296.368,E2 20296.368} C_VEL
LIN {X 0,Y 433.251,Z 286.266,A -85,B 0,C 180,E1 20292.545,E2 20292.545} C_VEL
LIN {X 0,Y 433.242,Z 286.267,A -85,B 0,C 180,E1 20288.735,E2 20288.735} C_VEL
LIN {X 0,Y 433.24,Z 286.266,A -85,B 0,C 180,E1 20284.913,E2 20284.913} C_VEL
LIN {X 0,Y 433.242,Z 286.265,A -85,B 0,C 180,E1 20281.106,E2 20281.106} C_VEL
LIN {X 0,Y 433.254,Z 286.263,A -85,B 0,C 180,E1 20277.315,E2 20277.315} C_VEL
LIN {X 0,Y 433.259,Z 286.263,A -85,B 0,C 180,E1 20273.53,E2 20273.53} C_VEL
LIN {X 0,Y 433.256,Z 286.264,A -85,B 0,C 180,E1 20269.683,E2 20269.683} C_VEL
LIN {X 0,Y 433.255,Z 286.265,A -85,B 0,C 180,E1 20265.802,E2 20265.802} C_VEL
LIN {X 0,Y 433.254,Z 286.265,A -85,B 0,C 180,E1 20261.987,E2 20261.987} C_VEL
LIN {X 0,Y 433.258,Z 286.265,A -85,B 0,C 180,E1 20258.092,E2 20258.092} C_VEL
LIN {X 0,Y 433.25,Z 286.266,A -85,B 0,C 180,E1 20254.235,E2 20254.235} C_VEL
LIN {X 0,Y 433.253,Z 286.269,A -85,B 0,C 180,E1 20251.807,E2 20251.807} C_VEL
LIN {X 0,Y 432.26,Z 286.388,A -85,B 0,C 180,E1 20250.788,E2 20250.788} C_VEL
LIN {X 0,Y 425.743,Z 287.203,A -85,B 0,C 180,E1 20247.844,E2 20247.844} C_VEL
LIN {X 0,Y 425.312,Z 287.253,A -85,B 0,C 180,E1 20247.17,E2 20247.17} C_VEL
LIN {X 0,Y 425.309,Z 287.254,A -85,B 0,C 180,E1 20243.385,E2 20243.385} C_VEL
LIN {X 0,Y 425.308,Z 287.255,A -85,B 0,C 180,E1 20239.571,E2 20239.571} C_VEL
LIN {X 0,Y 425.316,Z 287.254,A -85,B 0,C 180,E1 20235.71,E2 20235.71} C_VEL
LIN {X 0,Y 425.317,Z 287.254,A -85,B 0,C 180,E1 20231.922,E2 20231.922} C_VEL
LIN {X 0,Y 425.319,Z 287.254,A -85,B 0,C 180,E1 20228.051,E2 20228.051} C_VEL
LIN {X 0,Y 425.319,Z 287.253,A -85,B 0,C 180,E1 20224.207,E2 20224.207} C_VEL
LIN {X 0,Y 425.323,Z 287.253,A -85,B 0,C 180,E1 20220.419,E2 20220.419} C_VEL
LIN {X 0,Y 425.315,Z 287.255,A -85,B 0,C 180,E1 20216.57,E2 20216.57} C_VEL
LIN {X 0,Y 425.3,Z 287.256,A -85,B 0,C 180,E1 20212.83,E2 20212.83} C_VEL
LIN {X 0,Y 425.297,Z 287.257,A -85,B 0,C 180,E1 20208.995,E2 20208.995} C_VEL
LIN {X 0,Y 425.301,Z 287.256,A -85,B 0,C 180,E1 20205.149,E2 20205.149} C_VEL
LIN {X 0,Y 425.311,Z 287.255,A -85,B 0,C 180,E1 20201.345,E2 20201.345} C_VEL
LIN {X 0,Y 425.317,Z 287.254,A -85,B 0,C 180,E1 20197.508,E2 20197.508} C_VEL
LIN {X 0,Y 425.321,Z 287.254,A -85,B 0,C 180,E1 20193.678,E2 20193.678} C_VEL
LIN {X 0,Y 425.327,Z 287.254,A -85,B 0,C 180,E1 20189.84,E2 20189.84} C_VEL
LIN {X 0,Y 425.308,Z 287.257,A -85,B 0,C 180,E1 20186.08,E2 20186.08} C_VEL
LIN {X 0,Y 425.296,Z 287.258,A -85,B 0,C 180,E1 20182.241,E2 20182.241} C_VEL
LIN {X 0,Y 425.287,Z 287.26,A -85,B 0,C 180,E1 20178.505,E2 20178.505} C_VEL
LIN {X 0,Y 425.283,Z 287.232,A -85,B 0,C 180,E1 20174.709,E2 20174.709} C_VEL
LIN {X 0,Y 425.298,Z 287.238,A -85,B 0,C 180,E1 20170.978,E2 20170.978} C_VEL
LIN {X 0,Y 425.318,Z 287.252,A -85,B 0,C 180,E1 20167.157,E2 20167.157} C_VEL
LIN {X 0,Y 425.312,Z 287.22,A -85,B 0,C 180,E1 20163.369,E2 20163.369} C_VEL
LIN {X 0,Y 425.306,Z 287.255,A -85,B 0,C 180,E1 20159.596,E2 20159.596} C_VEL
LIN {X 0,Y 425.282,Z 287.239,A -85,B 0,C 180,E1 20155.82,E2 20155.82} C_VEL
LIN {X 0,Y 425.271,Z 287.237,A -85,B 0,C 180,E1 20152.163,E2 20152.163} C_VEL
LIN {X 0,Y 425.275,Z 287.262,A -85,B 0,C 180,E1 20148.335,E2 20148.335} C_VEL
LIN {X 0,Y 425.281,Z 287.229,A -85,B 0,C 180,E1 20144.559,E2 20144.559} C_VEL
LIN {X 0,Y 425.304,Z 287.239,A -85,B 0,C 180,E1 20140.784,E2 20140.784} C_VEL
LIN {X 0,Y 425.316,Z 287.258,A -85,B 0,C 180,E1 20136.884,E2 20136.884} C_VEL
LIN {X 0,Y 425.31,Z 287.239,A -85,B 0,C 180,E1 20132.995,E2 20132.995} C_VEL
LIN {X 0,Y 425.28,Z 287.243,A -85,B 0,C 180,E1 20129.324,E2 20129.324} C_VEL
LIN {X 0,Y 425.262,Z 287.249,A -85,B 0,C 180,E1 20125.612,E2 20125.612} C_VEL
LIN {X 0,Y 425.295,Z 287.403,A -85,B 0,C 180,E1 20122.238,E2 20122.238} C_VEL
LIN {X 0,Y 429.73,Z 299.238,A -85,B 0,C 180,E1 20119.259,E2 20119.259} C_VEL
LIN {X 0,Y 434.944,Z 307.467,A -85,B 0,C 180,E1 20118.213,E2 20118.213} C_VEL
LIN {X 0,Y 445.606,Z 324.282,A -85,B 0,C 180,E1 20116.328,E2 20116.328} C_VEL
LIN {X 0,Y 457.868,Z 345.552,A -85,B 0,C 180,E1 20114.298,E2 20114.298} C_VEL
LIN {X 0,Y 460.956,Z 351.701,A -85,B 0,C 180,E1 20113.798,E2 20113.798} C_VEL
LIN {X 0,Y 454.935,Z 565.269,A -85,B 0,C 180,E1 20110.073,E2 20110.073} C_VEL
LIN {X 0,Y 453.578,Z 608.101,A -85,B 0,C 180,E1 20109.294,E2 20109.294} C_VEL
LIN {X 0,Y 452.025,Z 630.3,A -85,B 0,C 180,E1 20108.679,E2 20108.679} C_VEL
LIN {X 0,Y 450.453,Z 647.913,A -85,B 0,C 180,E1 20108.02,E2 20108.02} C_VEL
LIN {X 0,Y 448.539,Z 666.218,A -85,B 0,C 180,E1 20107.163,E2 20107.163} C_VEL
LIN {X 0,Y 445.856,Z 687.757,A -85,B 0,C 180,E1 20105.903,E2 20105.903} C_VEL
LIN {X 0,Y 443.371,Z 705.542,A -85,B 0,C 180,E1 20104.63,E2 20104.63} C_VEL
LIN {X 0,Y 440.776,Z 723.242,A -85,B 0,C 180,E1 20103.139,E2 20103.139} C_VEL
LIN {X 0,Y 437.839,Z 741.599,A -85,B 0,C 180,E1 20101.299,E2 20101.299} C_VEL
LIN {X 0,Y 435.452,Z 756.312,A -85,B 0,C 180,E1 20099.581,E2 20099.581} C_VEL
LIN {X 0,Y 432.97,Z 771.799,A -85,B 0,C 180,E1 20097.506,E2 20097.506} C_VEL
LIN {X 0,Y 430.53,Z 787.12,A -85,B 0,C 180,E1 20095.078,E2 20095.078} C_VEL
LIN {X 0,Y 428.867,Z 798.189,A -85,B 0,C 180,E1 20093.058,E2 20093.058} C_VEL
LIN {X 0,Y 427.243,Z 810.173,A -85,B 0,C 180,E1 20090.55,E2 20090.55} C_VEL
LIN {X 0,Y 425.899,Z 821.225,A -85,B 0,C 180,E1 20087.769,E2 20087.769} C_VEL
LIN {X 0,Y 425.096,Z 829.153,A -85,B 0,C 180,E1 20085.413,E2 20085.413} C_VEL
LIN {X 0,Y 424.483,Z 836.935,A -85,B 0,C 180,E1 20082.653,E2 20082.653} C_VEL
LIN {X 0,Y 424.125,Z 843.176,A -85,B 0,C 180,E1 20079.772,E2 20079.772} C_VEL
LIN {X 0,Y 423.986,Z 847.038,A -85,B 0,C 180,E1 20077.452,E2 20077.452} C_VEL
LIN {X 0,Y 423.928,Z 849.982,A -85,B 0,C 180,E1 20075.006,E2 20075.006} C_VEL
LIN {X 0,Y 423.908,Z 852.027,A -85,B 0,C 180,E1 20072.163,E2 20072.163} C_VEL
LIN {X 0,Y 423.9,Z 852.352,A -85,B 0,C 180,E1 20069.324,E2 20069.324} C_VEL
LIN {X 0,Y 423.914,Z 851.455,A -85,B 0,C 180,E1 20066.89,E2 20066.89} C_VEL
LIN {X 0,Y 423.936,Z 849.416,A -85,B 0,C 180,E1 20064.436,E2 20064.436} C_VEL
LIN {X 0,Y 424.037,Z 845.673,A -85,B 0,C 180,E1 20061.594,E2 20061.594} C_VEL
LIN {X 0,Y 424.276,Z 840.079,A -85,B 0,C 180,E1 20058.721,E2 20058.721} C_VEL
LIN {X 0,Y 424.656,Z 834.345,A -85,B 0,C 180,E1 20056.382,E2 20056.382} C_VEL
LIN {X 0,Y 425.302,Z 826.988,A -85,B 0,C 180,E1 20053.895,E2 20053.895} C_VEL
LIN {X 0,Y 426.443,Z 816.487,A -85,B 0,C 180,E1 20050.98,E2 20050.98} C_VEL
LIN {X 0,Y 427.733,Z 806.328,A -85,B 0,C 180,E1 20048.614,E2 20048.614} C_VEL
LIN {X 0,Y 429.53,Z 793.875,A -85,B 0,C 180,E1 20046.107,E2 20046.107} C_VEL
LIN {X 0,Y 431.718,Z 779.523,A -85,B 0,C 180,E1 20043.674,E2 20043.674} C_VEL
LIN {X 0,Y 433.746,Z 766.819,A -85,B 0,C 180,E1 20041.8,E2 20041.8} C_VEL
LIN {X 0,Y 436.396,Z 750.772,A -85,B 0,C 180,E1 20039.732,E2 20039.732} C_VEL
LIN {X 0,Y 439.199,Z 733.084,A -85,B 0,C 180,E1 20037.812,E2 20037.812} C_VEL
LIN {X 0,Y 441.56,Z 717.837,A -85,B 0,C 180,E1 20036.384,E2 20036.384} C_VEL
LIN {X 0,Y 444.297,Z 699.453,A -85,B 0,C 180,E1 20034.903,E2 20034.903} C_VEL
LIN {X 0,Y 446.953,Z 679.205,A -85,B 0,C 180,E1 20033.564,E2 20033.564} C_VEL
LIN {X 0,Y 448.96,Z 662.259,A -85,B 0,C 180,E1 20032.638,E2 20032.638} C_VEL
LIN {X 0,Y 450.906,Z 643.21,A -85,B 0,C 180,E1 20031.782,E2 20031.782} C_VEL
LIN {X 0,Y 452.782,Z 620.409,A -85,B 0,C 180,E1 20031.02,E2 20031.02} C_VEL
LIN {X 0,Y 453.867,Z 601.467,A -85,B 0,C 180,E1 20030.573,E2 20030.573} C_VEL
LIN {X 0,Y 459.946,Z 386.548,A -85,B 0,C 180,E1 20026.815,E2 20026.815} C_VEL
LIN {X 0,Y 460.811,Z 351.044,A -85,B 0,C 180,E1 20026.171,E2 20026.171} C_VEL
LIN {X 0,Y 448.797,Z 329.557,A -85,B 0,C 180,E1 20024.212,E2 20024.212} C_VEL
LIN {X 0,Y 437.455,Z 311.251,A -85,B 0,C 180,E1 20022.242,E2 20022.242} C_VEL
LIN {X 0,Y 429.911,Z 299.628,A -85,B 0,C 180,E1 20020.808,E2 20020.808} C_VEL
LIN {X 0,Y 426.126,Z 289.964,A -85,B 0,C 180,E1 20018.447,E2 20018.447} C_VEL
LIN {X 0,Y 425.287,Z 287.315,A -85,B 0,C 180,E1 20017.681,E2 20017.681} C_VEL
LIN {X 0,Y 425.264,Z 287.246,A -85,B 0,C 180,E1 20013.908,E2 20013.908} C_VEL
LIN {X 0,Y 425.263,Z 287.243,A -85,B 0,C 180,E1 20010.094,E2 20010.094} C_VEL
LIN {X 0,Y 425.264,Z 287.234,A -85,B 0,C 180,E1 20006.232,E2 20006.232} C_VEL
LIN {X 0,Y 425.277,Z 287.255,A -85,B 0,C 180,E1 20002.49,E2 20002.49} C_VEL
LIN {X 0,Y 425.306,Z 287.244,A -85,B 0,C 180,E1 19998.788,E2 19998.788} C_VEL
LIN {X 0,Y 425.319,Z 287.22,A -85,B 0,C 180,E1 19994.946,E2 19994.946} C_VEL
LIN {X 0,Y 425.303,Z 287.248,A -85,B 0,C 180,E1 19991.115,E2 19991.115} C_VEL
LIN {X 0,Y 425.29,Z 287.245,A -85,B 0,C 180,E1 19987.294,E2 19987.294} C_VEL
LIN {X 0,Y 425.276,Z 287.229,A -85,B 0,C 180,E1 19983.505,E2 19983.505} C_VEL
LIN {X 0,Y 425.277,Z 287.26,A -85,B 0,C 180,E1 19979.731,E2 19979.731} C_VEL
LIN {X 0,Y 425.281,Z 287.227,A -85,B 0,C 180,E1 19975.955,E2 19975.955} C_VEL
LIN {X 0,Y 425.299,Z 287.247,A -85,B 0,C 180,E1 19972.163,E2 19972.163} C_VEL
LIN {X 0,Y 425.313,Z 287.249,A -85,B 0,C 180,E1 19968.336,E2 19968.336} C_VEL
LIN {X 0,Y 425.322,Z 287.222,A -85,B 0,C 180,E1 19964.539,E2 19964.539} C_VEL
LIN {X 0,Y 425.318,Z 287.258,A -85,B 0,C 180,E1 19960.642,E2 19960.642} C_VEL
LIN {X 0,Y 425.31,Z 287.259,A -85,B 0,C 180,E1 19956.806,E2 19956.806} C_VEL
LIN {X 0,Y 425.3,Z 287.259,A -85,B 0,C 180,E1 19952.997,E2 19952.997} C_VEL
LIN {X 0,Y 425.292,Z 287.26,A -85,B 0,C 180,E1 19949.169,E2 19949.169} C_VEL
LIN {X 0,Y 425.293,Z 287.26,A -85,B 0,C 180,E1 19945.324,E2 19945.324} C_VEL
LIN {X 0,Y 425.299,Z 287.259,A -85,B 0,C 180,E1 19941.464,E2 19941.464} C_VEL
LIN {X 0,Y 425.315,Z 287.257,A -85,B 0,C 180,E1 19937.752,E2 19937.752} C_VEL
LIN {X 0,Y 425.319,Z 287.257,A -85,B 0,C 180,E1 19933.906,E2 19933.906} C_VEL
LIN {X 0,Y 425.321,Z 287.256,A -85,B 0,C 180,E1 19930.099,E2 19930.099} C_VEL
LIN {X 0,Y 425.317,Z 287.256,A -85,B 0,C 180,E1 19926.26,E2 19926.26} C_VEL
LIN {X 0,Y 425.313,Z 287.256,A -85,B 0,C 180,E1 19922.411,E2 19922.411} C_VEL
LIN {X 0,Y 425.306,Z 287.256,A -85,B 0,C 180,E1 19918.658,E2 19918.658} C_VEL
LIN {X 0,Y 425.304,Z 287.256,A -85,B 0,C 180,E1 19914.844,E2 19914.844} C_VEL
LIN {X 0,Y 425.307,Z 287.257,A -85,B 0,C 180,E1 19910.936,E2 19910.936} C_VEL
LIN {X 0,Y 425.312,Z 287.258,A -85,B 0,C 180,E1 19907.089,E2 19907.089} C_VEL
LIN {X 0,Y 425.319,Z 287.257,A -85,B 0,C 180,E1 19903.283,E2 19903.283} C_VEL
LIN {X 0,Y 425.318,Z 287.258,A -85,B 0,C 180,E1 19899.335,E2 19899.335} C_VEL
LIN {X 0,Y 425.311,Z 287.258,A -85,B 0,C 180,E1 19895.531,E2 19895.531} C_VEL
LIN {X 0,Y 425.313,Z 287.256,A -85,B 0,C 180,E1 19891.617,E2 19891.617} C_VEL
LIN {X 0,Y 425.315,Z 287.256,A -85,B 0,C 180,E1 19887.844,E2 19887.844} C_VEL
LIN {X 0,Y 425.312,Z 287.253,A -85,B 0,C 180,E1 19887.17,E2 19887.17} C_VEL
LIN {X 0,Y 424.331,Z 287.381,A -85,B 0,C 180,E1 19886.132,E2 19886.132} C_VEL
LIN {X 0,Y 417.812,Z 288.191,A -85,B 0,C 180,E1 19883.132,E2 19883.132} C_VEL
LIN {X 0,Y 417.374,Z 288.248,A -85,B 0,C 180,E1 19882.445,E2 19882.445} C_VEL
LIN {X 0,Y 417.376,Z 288.246,A -85,B 0,C 180,E1 19878.532,E2 19878.532} C_VEL
LIN {X 0,Y 417.382,Z 288.243,A -85,B 0,C 180,E1 19874.58,E2 19874.58} C_VEL
LIN {X 0,Y 417.377,Z 288.243,A -85,B 0,C 180,E1 19870.696,E2 19870.696} C_VEL
LIN {X 0,Y 417.371,Z 288.243,A -85,B 0,C 180,E1 19866.867,E2 19866.867} C_VEL
LIN {X 0,Y 417.366,Z 288.243,A -85,B 0,C 180,E1 19863.021,E2 19863.021} C_VEL
LIN {X 0,Y 417.362,Z 288.244,A -85,B 0,C 180,E1 19859.159,E2 19859.159} C_VEL
LIN {X 0,Y 417.365,Z 288.244,A -85,B 0,C 180,E1 19855.239,E2 19855.239} C_VEL
LIN {X 0,Y 417.368,Z 288.243,A -85,B 0,C 180,E1 19851.35,E2 19851.35} C_VEL
LIN {X 0,Y 417.374,Z 288.243,A -85,B 0,C 180,E1 19847.504,E2 19847.504} C_VEL
LIN {X 0,Y 417.379,Z 288.242,A -85,B 0,C 180,E1 19843.624,E2 19843.624} C_VEL
LIN {X 0,Y 417.384,Z 288.242,A -85,B 0,C 180,E1 19839.741,E2 19839.741} C_VEL
LIN {X 0,Y 417.38,Z 288.244,A -85,B 0,C 180,E1 19835.936,E2 19835.936} C_VEL
LIN {X 0,Y 417.377,Z 288.245,A -85,B 0,C 180,E1 19832.004,E2 19832.004} C_VEL
LIN {X 0,Y 417.369,Z 288.247,A -85,B 0,C 180,E1 19828.16,E2 19828.16} C_VEL
LIN {X 0,Y 417.355,Z 288.247,A -85,B 0,C 180,E1 19824.334,E2 19824.334} C_VEL
LIN {X 0,Y 417.349,Z 288.247,A -85,B 0,C 180,E1 19820.474,E2 19820.474} C_VEL
LIN {X 0,Y 417.342,Z 288.223,A -85,B 0,C 180,E1 19816.565,E2 19816.565} C_VEL
LIN {X 0,Y 417.35,Z 288.249,A -85,B 0,C 180,E1 19812.733,E2 19812.733} C_VEL
LIN {X 0,Y 417.358,Z 288.213,A -85,B 0,C 180,E1 19808.958,E2 19808.958} C_VEL
LIN {X 0,Y 417.375,Z 288.23,A -85,B 0,C 180,E1 19805.223,E2 19805.223} C_VEL
LIN {X 0,Y 417.383,Z 288.236,A -85,B 0,C 180,E1 19801.235,E2 19801.235} C_VEL
LIN {X 0,Y 417.372,Z 288.208,A -85,B 0,C 180,E1 19797.36,E2 19797.36} C_VEL
LIN {X 0,Y 417.362,Z 288.246,A -85,B 0,C 180,E1 19793.535,E2 19793.535} C_VEL
LIN {X 0,Y 417.339,Z 288.225,A -85,B 0,C 180,E1 19789.788,E2 19789.788} C_VEL
LIN {X 0,Y 417.328,Z 288.223,A -85,B 0,C 180,E1 19785.997,E2 19785.997} C_VEL
LIN {X 0,Y 417.332,Z 288.25,A -85,B 0,C 180,E1 19782.142,E2 19782.142} C_VEL
LIN {X 0,Y 417.333,Z 288.226,A -85,B 0,C 180,E1 19778.349,E2 19778.349} C_VEL
LIN {X 0,Y 417.352,Z 288.218,A -85,B 0,C 180,E1 19774.607,E2 19774.607} C_VEL
LIN {X 0,Y 417.371,Z 288.232,A -85,B 0,C 180,E1 19770.745,E2 19770.745} C_VEL
LIN {X 0,Y 417.367,Z 288.233,A -85,B 0,C 180,E1 19766.893,E2 19766.893} C_VEL
LIN {X 0,Y 417.372,Z 288.492,A -85,B 0,C 180,E1 19763.303,E2 19763.303} C_VEL
LIN {X 0,Y 421.522,Z 299.148,A -85,B 0,C 180,E1 19760.528,E2 19760.528} C_VEL
LIN {X 0,Y 434.238,Z 318.547,A -85,B 0,C 180,E1 19758.048,E2 19758.048} C_VEL
LIN {X 0,Y 446.252,Z 338.599,A -85,B 0,C 180,E1 19755.917,E2 19755.917} C_VEL
LIN {X 0,Y 455.087,Z 354.569,A -85,B 0,C 180,E1 19754.443,E2 19754.443} C_VEL
LIN {X 0,Y 448.72,Z 568.462,A -85,B 0,C 180,E1 19750.673,E2 19750.673} C_VEL
LIN {X 0,Y 447.345,Z 608.841,A -85,B 0,C 180,E1 19749.926,E2 19749.926} C_VEL
LIN {X 0,Y 445.706,Z 630.652,A -85,B 0,C 180,E1 19749.306,E2 19749.306} C_VEL
LIN {X 0,Y 444.024,Z 648.523,A -85,B 0,C 180,E1 19748.626,E2 19748.626} C_VEL
LIN {X 0,Y 441.807,Z 668.606,A -85,B 0,C 180,E1 19747.663,E2 19747.663} C_VEL
LIN {X 0,Y 439.133,Z 688.492,A -85,B 0,C 180,E1 19746.459,E2 19746.459} C_VEL
LIN {X 0,Y 436.659,Z 705.287,A -85,B 0,C 180,E1 19745.241,E2 19745.241} C_VEL
LIN {X 0,Y 433.858,Z 723.346,A -85,B 0,C 180,E1 19743.7,E2 19743.7} C_VEL
LIN {X 0,Y 430.703,Z 741.96,A -85,B 0,C 180,E1 19741.8,E2 19741.8} C_VEL
LIN {X 0,Y 428.178,Z 756.609,A -85,B 0,C 180,E1 19740.058,E2 19740.058} C_VEL
LIN {X 0,Y 425.477,Z 772.527,A -85,B 0,C 180,E1 19737.881,E2 19737.881} C_VEL
LIN {X 0,Y 422.96,Z 787.275,A -85,B 0,C 180,E1 19735.482,E2 19735.482} C_VEL
LIN {X 0,Y 421.142,Z 798.65,A -85,B 0,C 180,E1 19733.358,E2 19733.358} C_VEL
LIN {X 0,Y 419.339,Z 811.122,A -85,B 0,C 180,E1 19730.663,E2 19730.663} C_VEL
LIN {X 0,Y 418,Z 821.467,A -85,B 0,C 180,E1 19727.972,E2 19727.972} C_VEL
LIN {X 0,Y 417.133,Z 829.518,A -85,B 0,C 180,E1 19725.511,E2 19725.511} C_VEL
LIN {X 0,Y 416.455,Z 837.657,A -85,B 0,C 180,E1 19722.478,E2 19722.478} C_VEL
LIN {X 0,Y 416.13,Z 843.175,A -85,B 0,C 180,E1 19719.822,E2 19719.822} C_VEL
LIN {X 0,Y 415.987,Z 846.982,A -85,B 0,C 180,E1 19717.457,E2 19717.457} C_VEL
LIN {X 0,Y 415.926,Z 850.007,A -85,B 0,C 180,E1 19714.826,E2 19714.826} C_VEL
LIN {X 0,Y 415.904,Z 851.883,A -85,B 0,C 180,E1 19711.791,E2 19711.791} C_VEL
LIN {X 0,Y 415.908,Z 852.076,A -85,B 0,C 180,E1 19709.174,E2 19709.174} C_VEL
LIN {X 0,Y 415.916,Z 851.123,A -85,B 0,C 180,E1 19706.693,E2 19706.693} C_VEL
LIN {X 0,Y 415.939,Z 849.043,A -85,B 0,C 180,E1 19704.206,E2 19704.206} C_VEL
LIN {X 0,Y 416.048,Z 844.932,A -85,B 0,C 180,E1 19701.153,E2 19701.153} C_VEL
LIN {X 0,Y 416.307,Z 839.809,A -85,B 0,C 180,E1 19698.494,E2 19698.494} C_VEL
LIN {X 0,Y 416.72,Z 834.091,A -85,B 0,C 180,E1 19696.118,E2 19696.118} C_VEL
LIN {X 0,Y 417.417,Z 826.733,A -85,B 0,C 180,E1 19693.582,E2 19693.582} C_VEL
LIN {X 0,Y 418.649,Z 816.231,A -85,B 0,C 180,E1 19690.612,E2 19690.612} C_VEL
LIN {X 0,Y 420.031,Z 806.071,A -85,B 0,C 180,E1 19688.202,E2 19688.202} C_VEL
LIN {X 0,Y 421.835,Z 794.336,A -85,B 0,C 180,E1 19685.792,E2 19685.792} C_VEL
LIN {X 0,Y 424.226,Z 779.701,A -85,B 0,C 180,E1 19683.246,E2 19683.246} C_VEL
LIN {X 0,Y 426.464,Z 766.5,A -85,B 0,C 180,E1 19681.265,E2 19681.265} C_VEL
LIN {X 0,Y 429.37,Z 750.03,A -85,B 0,C 180,E1 19679.116,E2 19679.116} C_VEL
LIN {X 0,Y 432.246,Z 732.828,A -85,B 0,C 180,E1 19677.23,E2 19677.23} C_VEL
LIN {X 0,Y 434.872,Z 716.811,A -85,B 0,C 180,E1 19675.717,E2 19675.717} C_VEL
LIN {X 0,Y 437.93,Z 697.29,A -85,B 0,C 180,E1 19674.146,E2 19674.146} C_VEL
LIN {X 0,Y 440.57,Z 677.818,A -85,B 0,C 180,E1 19672.867,E2 19672.867} C_VEL
LIN {X 0,Y 442.77,Z 660.026,A -85,B 0,C 180,E1 19671.9,E2 19671.9} C_VEL
LIN {X 0,Y 445.1,Z 637.878,A -85,B 0,C 180,E1 19670.943,E2 19670.943} C_VEL
LIN {X 0,Y 446.693,Z 618.236,A -85,B 0,C 180,E1 19670.32,E2 19670.32} C_VEL
LIN {X 0,Y 447.767,Z 599.549,A -85,B 0,C 180,E1 19669.887,E2 19669.887} C_VEL
LIN {X 0,Y 454.26,Z 381.55,A -85,B 0,C 180,E1 19666.036,E2 19666.036} C_VEL
LIN {X 0,Y 454.962,Z 354.328,A -85,B 0,C 180,E1 19665.536,E2 19665.536} C_VEL
LIN {X 0,Y 443.994,Z 334.63,A -85,B 0,C 180,E1 19663.693,E2 19663.693} C_VEL
LIN {X 0,Y 433.159,Z 316.916,A -85,B 0,C 180,E1 19661.755,E2 19661.755} C_VEL
LIN {X 0,Y 423.784,Z 302.888,A -85,B 0,C 180,E1 19659.966,E2 19659.966} C_VEL
LIN {X 0,Y 421.278,Z 298.543,A -85,B 0,C 180,E1 19659.367,E2 19659.367} C_VEL
LIN {X 0,Y 417.344,Z 288.343,A -85,B 0,C 180,E1 19656.623,E2 19656.623} C_VEL
LIN {X 0,Y 417.357,Z 288.236,A -85,B 0,C 180,E1 19652.944,E2 19652.944} C_VEL
LIN {X 0,Y 417.378,Z 288.235,A -85,B 0,C 180,E1 19649.031,E2 19649.031} C_VEL
LIN {X 0,Y 417.37,Z 288.217,A -85,B 0,C 180,E1 19645.089,E2 19645.089} C_VEL
LIN {X 0,Y 417.359,Z 288.215,A -85,B 0,C 180,E1 19641.268,E2 19641.268} C_VEL
LIN {X 0,Y 417.348,Z 288.246,A -85,B 0,C 180,E1 19637.426,E2 19637.426} C_VEL
LIN {X 0,Y 417.33,Z 288.225,A -85,B 0,C 180,E1 19633.721,E2 19633.721} C_VEL
LIN {X 0,Y 417.331,Z 288.22,A -85,B 0,C 180,E1 19629.933,E2 19629.933} C_VEL
LIN {X 0,Y 417.34,Z 288.249,A -85,B 0,C 180,E1 19626.051,E2 19626.051} C_VEL
LIN {X 0,Y 417.348,Z 288.214,A -85,B 0,C 180,E1 19622.197,E2 19622.197} C_VEL
LIN {X 0,Y 417.374,Z 288.234,A -85,B 0,C 180,E1 19618.49,E2 19618.49} C_VEL
LIN {X 0,Y 417.377,Z 288.235,A -85,B 0,C 180,E1 19614.501,E2 19614.501} C_VEL
LIN {X 0,Y 417.375,Z 288.209,A -85,B 0,C 180,E1 19610.735,E2 19610.735} C_VEL
LIN {X 0,Y 417.373,Z 288.242,A -85,B 0,C 180,E1 19606.845,E2 19606.845} C_VEL
LIN {X 0,Y 417.358,Z 288.229,A -85,B 0,C 180,E1 19603.006,E2 19603.006} C_VEL
LIN {X 0,Y 417.352,Z 288.248,A -85,B 0,C 180,E1 19599.233,E2 19599.233} C_VEL
LIN {X 0,Y 417.351,Z 288.249,A -85,B 0,C 180,E1 19595.364,E2 19595.364} C_VEL
LIN {X 0,Y 417.356,Z 288.248,A -85,B 0,C 180,E1 19591.527,E2 19591.527} C_VEL
LIN {X 0,Y 417.364,Z 288.247,A -85,B 0,C 180,E1 19587.708,E2 19587.708} C_VEL
LIN {X 0,Y 417.373,Z 288.247,A -85,B 0,C 180,E1 19583.832,E2 19583.832} C_VEL
LIN {X 0,Y 417.385,Z 288.243,A -85,B 0,C 180,E1 19580.045,E2 19580.045} C_VEL
LIN {X 0,Y 417.382,Z 288.243,A -85,B 0,C 180,E1 19576.14,E2 19576.14} C_VEL
LIN {X 0,Y 417.38,Z 288.243,A -85,B 0,C 180,E1 19572.249,E2 19572.249} C_VEL
LIN {X 0,Y 417.384,Z 288.243,A -85,B 0,C 180,E1 19568.347,E2 19568.347} C_VEL
LIN {X 0,Y 417.377,Z 288.244,A -85,B 0,C 180,E1 19564.426,E2 19564.426} C_VEL
LIN {X 0,Y 417.374,Z 288.244,A -85,B 0,C 180,E1 19560.521,E2 19560.521} C_VEL
LIN {X 0,Y 417.368,Z 288.245,A -85,B 0,C 180,E1 19556.613,E2 19556.613} C_VEL
LIN {X 0,Y 417.365,Z 288.247,A -85,B 0,C 180,E1 19552.686,E2 19552.686} C_VEL
LIN {X 0,Y 417.369,Z 288.247,A -85,B 0,C 180,E1 19548.868,E2 19548.868} C_VEL
LIN {X 0,Y 417.375,Z 288.247,A -85,B 0,C 180,E1 19544.994,E2 19544.994} C_VEL
LIN {X 0,Y 417.377,Z 288.247,A -85,B 0,C 180,E1 19541.188,E2 19541.188} C_VEL
LIN {X 0,Y 417.379,Z 288.246,A -85,B 0,C 180,E1 19537.294,E2 19537.294} C_VEL
LIN {X 0,Y 417.372,Z 288.245,A -85,B 0,C 180,E1 19533.433,E2 19533.433} C_VEL
LIN {X 0,Y 417.371,Z 288.244,A -85,B 0,C 180,E1 19529.588,E2 19529.588} C_VEL
LIN {X 0,Y 417.373,Z 288.244,A -85,B 0,C 180,E1 19525.741,E2 19525.741} C_VEL
LIN {X 0,Y 417.374,Z 288.248,A -85,B 0,C 180,E1 19522.445,E2 19522.445} C_VEL
LIN {X 0,Y 416.391,Z 288.373,A -85,B 0,C 180,E1 19521.387,E2 19521.387} C_VEL
LIN {X 0,Y 409.885,Z 289.178,A -85,B 0,C 180,E1 19518.33,E2 19518.33} C_VEL
LIN {X 0,Y 409.433,Z 289.232,A -85,B 0,C 180,E1 19517.629,E2 19517.629} C_VEL
LIN {X 0,Y 409.439,Z 289.231,A -85,B 0,C 180,E1 19513.836,E2 19513.836} C_VEL
LIN {X 0,Y 409.439,Z 289.232,A -85,B 0,C 180,E1 19509.86,E2 19509.86} C_VEL
LIN {X 0,Y 409.441,Z 289.233,A -85,B 0,C 180,E1 19505.933,E2 19505.933} C_VEL
LIN {X 0,Y 409.441,Z 289.233,A -85,B 0,C 180,E1 19502.04,E2 19502.04} C_VEL
LIN {X 0,Y 409.442,Z 289.234,A -85,B 0,C 180,E1 19498.166,E2 19498.166} C_VEL
LIN {X 0,Y 409.44,Z 289.235,A -85,B 0,C 180,E1 19494.169,E2 19494.169} C_VEL
LIN {X 0,Y 409.445,Z 289.235,A -85,B 0,C 180,E1 19490.224,E2 19490.224} C_VEL
LIN {X 0,Y 409.438,Z 289.236,A -85,B 0,C 180,E1 19486.285,E2 19486.285} C_VEL
LIN {X 0,Y 409.431,Z 289.236,A -85,B 0,C 180,E1 19482.377,E2 19482.377} C_VEL
LIN {X 0,Y 409.422,Z 289.237,A -85,B 0,C 180,E1 19478.516,E2 19478.516} C_VEL
LIN {X 0,Y 409.416,Z 289.238,A -85,B 0,C 180,E1 19474.615,E2 19474.615} C_VEL
LIN {X 0,Y 409.414,Z 289.238,A -85,B 0,C 180,E1 19470.691,E2 19470.691} C_VEL
LIN {X 0,Y 409.413,Z 289.237,A -85,B 0,C 180,E1 19466.703,E2 19466.703} C_VEL
LIN {X 0,Y 409.415,Z 289.237,A -85,B 0,C 180,E1 19462.849,E2 19462.849} C_VEL
LIN {X 0,Y 409.42,Z 289.237,A -85,B 0,C 180,E1 19458.954,E2 19458.954} C_VEL
LIN {X 0,Y 409.429,Z 289.199,A -85,B 0,C 180,E1 19455.147,E2 19455.147} C_VEL
LIN {X 0,Y 409.434,Z 289.216,A -85,B 0,C 180,E1 19451.266,E2 19451.266} C_VEL
LIN {X 0,Y 409.449,Z 289.226,A -85,B 0,C 180,E1 19447.295,E2 19447.295} C_VEL
LIN {X 0,Y 409.433,Z 289.195,A -85,B 0,C 180,E1 19443.36,E2 19443.36} C_VEL
LIN {X 0,Y 409.441,Z 289.225,A -85,B 0,C 180,E1 19439.44,E2 19439.44} C_VEL
LIN {X 0,Y 409.423,Z 289.218,A -85,B 0,C 180,E1 19435.518,E2 19435.518} C_VEL
LIN {X 0,Y 409.404,Z 289.203,A -85,B 0,C 180,E1 19431.715,E2 19431.715} C_VEL
LIN {X 0,Y 409.399,Z 289.238,A -85,B 0,C 180,E1 19427.876,E2 19427.876} C_VEL
LIN {X 0,Y 409.39,Z 289.212,A -85,B 0,C 180,E1 19423.98,E2 19423.98} C_VEL
LIN {X 0,Y 409.389,Z 289.208,A -85,B 0,C 180,E1 19420.096,E2 19420.096} C_VEL
LIN {X 0,Y 409.395,Z 289.236,A -85,B 0,C 180,E1 19416.236,E2 19416.236} C_VEL
LIN {X 0,Y 409.399,Z 289.232,A -85,B 0,C 180,E1 19412.353,E2 19412.353} C_VEL
LIN {X 0,Y 409.423,Z 289.226,A -85,B 0,C 180,E1 19408.656,E2 19408.656} C_VEL
LIN {X 0,Y 409.428,Z 289.239,A -85,B 0,C 180,E1 19404.807,E2 19404.807} C_VEL
LIN {X 0,Y 409.455,Z 289.545,A -85,B 0,C 180,E1 19404.467,E2 19404.467} C_VEL
LIN {X 0,Y 412.84,Z 298.393,A -85,B 0,C 180,E1 19402.036,E2 19402.036} C_VEL
LIN {X 0,Y 418.452,Z 306.818,A -85,B 0,C 180,E1 19400.802,E2 19400.802} C_VEL
LIN {X 0,Y 426.66,Z 319.123,A -85,B 0,C 180,E1 19399.17,E2 19399.17} C_VEL
LIN {X 0,Y 436.932,Z 335.76,A -85,B 0,C 180,E1 19397.251,E2 19397.251} C_VEL
LIN {X 0,Y 448.483,Z 356.222,A -85,B 0,C 180,E1 19395.234,E2 19395.234} C_VEL
LIN {X 0,Y 449.253,Z 358.217,A -85,B 0,C 180,E1 19395.091,E2 19395.091} C_VEL
LIN {X 0,Y 442.535,Z 572.292,A -85,B 0,C 180,E1 19391.279,E2 19391.279} C_VEL
LIN {X 0,Y 441.175,Z 609.283,A -85,B 0,C 180,E1 19390.58,E2 19390.58} C_VEL
LIN {X 0,Y 439.46,Z 630.81,A -85,B 0,C 180,E1 19389.958,E2 19389.958} C_VEL
LIN {X 0,Y 437.661,Z 648.976,A -85,B 0,C 180,E1 19389.257,E2 19389.257} C_VEL
LIN {X 0,Y 435.239,Z 669.741,A -85,B 0,C 180,E1 19388.242,E2 19388.242} C_VEL
LIN {X 0,Y 432.453,Z 689.226,A -85,B 0,C 180,E1 19387.033,E2 19387.033} C_VEL
LIN {X 0,Y 429.821,Z 706.169,A -85,B 0,C 180,E1 19385.78,E2 19385.78} C_VEL
LIN {X 0,Y 426.732,Z 724.997,A -85,B 0,C 180,E1 19384.135,E2 19384.135} C_VEL
LIN {X 0,Y 423.627,Z 742.189,A -85,B 0,C 180,E1 19382.332,E2 19382.332} C_VEL
LIN {X 0,Y 420.936,Z 756.906,A -85,B 0,C 180,E1 19380.551,E2 19380.551} C_VEL
LIN {X 0,Y 417.993,Z 773.178,A -85,B 0,C 180,E1 19378.269,E2 19378.269} C_VEL
LIN {X 0,Y 415.481,Z 787.017,A -85,B 0,C 180,E1 19375.975,E2 19375.975} C_VEL
LIN {X 0,Y 413.546,Z 798.393,A -85,B 0,C 180,E1 19373.813,E2 19373.813} C_VEL
LIN {X 0,Y 411.609,Z 810.865,A -85,B 0,C 180,E1 19371.07,E2 19371.07} C_VEL
LIN {X 0,Y 410.168,Z 821.211,A -85,B 0,C 180,E1 19368.328,E2 19368.328} C_VEL
LIN {X 0,Y 409.25,Z 829.076,A -85,B 0,C 180,E1 19365.88,E2 19365.88} C_VEL
LIN {X 0,Y 408.524,Z 837.094,A -85,B 0,C 180,E1 19362.869,E2 19362.869} C_VEL
LIN {X 0,Y 408.142,Z 842.953,A -85,B 0,C 180,E1 19360,E2 19360} C_VEL
LIN {X 0,Y 407.988,Z 846.925,A -85,B 0,C 180,E1 19357.463,E2 19357.463} C_VEL
LIN {X 0,Y 407.925,Z 850.033,A -85,B 0,C 180,E1 19354.639,E2 19354.639} C_VEL
LIN {X 0,Y 407.908,Z 851.69,A -85,B 0,C 180,E1 19351.545,E2 19351.545} C_VEL
LIN {X 0,Y 407.916,Z 851.801,A -85,B 0,C 180,E1 19349.017,E2 19349.017} C_VEL
LIN {X 0,Y 407.918,Z 850.875,A -85,B 0,C 180,E1 19346.628,E2 19346.628} C_VEL
LIN {X 0,Y 407.942,Z 848.794,A -85,B 0,C 180,E1 19344.092,E2 19344.092} C_VEL
LIN {X 0,Y 408.06,Z 844.681,A -85,B 0,C 180,E1 19340.978,E2 19340.978} C_VEL
LIN {X 0,Y 408.34,Z 839.574,A -85,B 0,C 180,E1 19338.274,E2 19338.274} C_VEL
LIN {X 0,Y 408.79,Z 833.837,A -85,B 0,C 180,E1 19335.843,E2 19335.843} C_VEL
LIN {X 0,Y 409.596,Z 826.044,A -85,B 0,C 180,E1 19333.113,E2 19333.113} C_VEL
LIN {X 0,Y 410.947,Z 815.407,A -85,B 0,C 180,E1 19330.085,E2 19330.085} C_VEL
LIN {X 0,Y 412.35,Z 805.814,A -85,B 0,C 180,E1 19327.774,E2 19327.774} C_VEL
LIN {X 0,Y 414.41,Z 793.359,A -85,B 0,C 180,E1 19325.178,E2 19325.178} C_VEL
LIN {X 0,Y 416.833,Z 779.444,A -85,B 0,C 180,E1 19322.733,E2 19322.733} C_VEL
LIN {X 0,Y 419.206,Z 766.304,A -85,B 0,C 180,E1 19320.729,E2 19320.729} C_VEL
LIN {X 0,Y 422.203,Z 750.259,A -85,B 0,C 180,E1 19318.601,E2 19318.601} C_VEL
LIN {X 0,Y 425.346,Z 732.573,A -85,B 0,C 180,E1 19316.63,E2 19316.63} C_VEL
LIN {X 0,Y 428.119,Z 716.556,A -85,B 0,C 180,E1 19315.098,E2 19315.098} C_VEL
LIN {X 0,Y 431.318,Z 697.131,A -85,B 0,C 180,E1 19313.517,E2 19313.517} C_VEL
LIN {X 0,Y 434.11,Z 677.565,A -85,B 0,C 180,E1 19312.219,E2 19312.219} C_VEL
LIN {X 0,Y 436.422,Z 659.775,A -85,B 0,C 180,E1 19311.244,E2 19311.244} C_VEL
LIN {X 0,Y 438.867,Z 637.628,A -85,B 0,C 180,E1 19310.28,E2 19310.28} C_VEL
LIN {X 0,Y 440.541,Z 617.894,A -85,B 0,C 180,E1 19309.65,E2 19309.65} C_VEL
LIN {X 0,Y 441.663,Z 599.09,A -85,B 0,C 180,E1 19309.211,E2 19309.211} C_VEL
LIN {X 0,Y 448.509,Z 381.21,A -85,B 0,C 180,E1 19305.321,E2 19305.321} C_VEL
LIN {X 0,Y 449.162,Z 357.562,A -85,B 0,C 180,E1 19304.883,E2 19304.883} C_VEL
LIN {X 0,Y 438.555,Z 338.6,A -85,B 0,C 180,E1 19303.042,E2 19303.042} C_VEL
LIN {X 0,Y 428.895,Z 322.576,A -85,B 0,C 180,E1 19301.258,E2 19301.258} C_VEL
LIN {X 0,Y 419.988,Z 309.088,A -85,B 0,C 180,E1 19299.512,E2 19299.512} C_VEL
LIN {X 0,Y 415.959,Z 303.171,A -85,B 0,C 180,E1 19298.68,E2 19298.68} C_VEL
LIN {X 0,Y 412.653,Z 297.992,A -85,B 0,C 180,E1 19297.885,E2 19297.885} C_VEL
LIN {X 0,Y 409.43,Z 289.336,A -85,B 0,C 180,E1 19295.45,E2 19295.45} C_VEL
LIN {X 0,Y 409.41,Z 289.231,A -85,B 0,C 180,E1 19291.509,E2 19291.509} C_VEL
LIN {X 0,Y 409.391,Z 289.237,A -85,B 0,C 180,E1 19287.806,E2 19287.806} C_VEL
LIN {X 0,Y 409.391,Z 289.233,A -85,B 0,C 180,E1 19283.918,E2 19283.918} C_VEL
LIN {X 0,Y 409.387,Z 289.205,A -85,B 0,C 180,E1 19279.994,E2 19279.994} C_VEL
LIN {X 0,Y 409.393,Z 289.212,A -85,B 0,C 180,E1 19276.166,E2 19276.166} C_VEL
LIN {X 0,Y 409.409,Z 289.236,A -85,B 0,C 180,E1 19272.352,E2 19272.352} C_VEL
LIN {X 0,Y 409.418,Z 289.199,A -85,B 0,C 180,E1 19268.491,E2 19268.491} C_VEL
LIN {X 0,Y 409.437,Z 289.222,A -85,B 0,C 180,E1 19264.763,E2 19264.763} C_VEL
LIN {X 0,Y 409.447,Z 289.222,A -85,B 0,C 180,E1 19260.7,E2 19260.7} C_VEL
LIN {X 0,Y 409.43,Z 289.196,A -85,B 0,C 180,E1 19256.78,E2 19256.78} C_VEL
LIN {X 0,Y 409.439,Z 289.23,A -85,B 0,C 180,E1 19252.846,E2 19252.846} C_VEL
LIN {X 0,Y 409.428,Z 289.215,A -85,B 0,C 180,E1 19248.877,E2 19248.877} C_VEL
LIN {X 0,Y 409.412,Z 289.204,A -85,B 0,C 180,E1 19245.142,E2 19245.142} C_VEL
LIN {X 0,Y 409.411,Z 289.239,A -85,B 0,C 180,E1 19241.342,E2 19241.342} C_VEL
LIN {X 0,Y 409.41,Z 289.238,A -85,B 0,C 180,E1 19237.387,E2 19237.387} C_VEL
LIN {X 0,Y 409.413,Z 289.236,A -85,B 0,C 180,E1 19233.454,E2 19233.454} C_VEL
LIN {X 0,Y 409.418,Z 289.237,A -85,B 0,C 180,E1 19229.548,E2 19229.548} C_VEL
LIN {X 0,Y 409.424,Z 289.237,A -85,B 0,C 180,E1 19225.63,E2 19225.63} C_VEL
LIN {X 0,Y 409.44,Z 289.234,A -85,B 0,C 180,E1 19221.842,E2 19221.842} C_VEL
LIN {X 0,Y 409.443,Z 289.233,A -85,B 0,C 180,E1 19217.932,E2 19217.932} C_VEL
LIN {X 0,Y 409.442,Z 289.232,A -85,B 0,C 180,E1 19214.103,E2 19214.103} C_VEL
LIN {X 0,Y 409.444,Z 289.233,A -85,B 0,C 180,E1 19210.141,E2 19210.141} C_VEL
LIN {X 0,Y 409.441,Z 289.233,A -85,B 0,C 180,E1 19206.224,E2 19206.224} C_VEL
LIN {X 0,Y 409.437,Z 289.234,A -85,B 0,C 180,E1 19202.33,E2 19202.33} C_VEL
LIN {X 0,Y 409.438,Z 289.234,A -85,B 0,C 180,E1 19198.436,E2 19198.436} C_VEL
LIN {X 0,Y 409.431,Z 289.236,A -85,B 0,C 180,E1 19194.528,E2 19194.528} C_VEL
LIN {X 0,Y 409.427,Z 289.237,A -85,B 0,C 180,E1 19190.72,E2 19190.72} C_VEL
LIN {X 0,Y 409.431,Z 289.237,A -85,B 0,C 180,E1 19186.748,E2 19186.748} C_VEL
LIN {X 0,Y 409.432,Z 289.235,A -85,B 0,C 180,E1 19182.84,E2 19182.84} C_VEL
LIN {X 0,Y 409.434,Z 289.233,A -85,B 0,C 180,E1 19178.85,E2 19178.85} C_VEL
LIN {X 0,Y 409.438,Z 289.232,A -85,B 0,C 180,E1 19175.043,E2 19175.043} C_VEL
LIN {X 0,Y 409.44,Z 289.23,A -85,B 0,C 180,E1 19171.119,E2 19171.119} C_VEL
LIN {X 0,Y 409.434,Z 289.231,A -85,B 0,C 180,E1 19167.187,E2 19167.187} C_VEL
LIN {X 0,Y 409.433,Z 289.232,A -85,B 0,C 180,E1 19163.269,E2 19163.269} C_VEL
LIN {X 0,Y 409.43,Z 289.233,A -85,B 0,C 180,E1 19159.304,E2 19159.304} C_VEL
LIN {X 0,Y 409.433,Z 289.232,A -85,B 0,C 180,E1 19157.629,E2 19157.629} C_VEL
LIN {X 0,Y 408.427,Z 289.362,A -85,B 0,C 180,E1 19156.551,E2 19156.551} C_VEL
LIN {X 0,Y 401.93,Z 290.172,A -85,B 0,C 180,E1 19153.433,E2 19153.433} C_VEL
LIN {X 0,Y 401.499,Z 290.221,A -85,B 0,C 180,E1 19152.718,E2 19152.718} C_VEL
LIN {X 0,Y 401.503,Z 290.219,A -85,B 0,C 180,E1 19148.68,E2 19148.68} C_VEL
LIN {X 0,Y 401.498,Z 290.219,A -85,B 0,C 180,E1 19144.687,E2 19144.687} C_VEL
LIN {X 0,Y 401.493,Z 290.22,A -85,B 0,C 180,E1 19140.785,E2 19140.785} C_VEL
LIN {X 0,Y 401.489,Z 290.221,A -85,B 0,C 180,E1 19136.8,E2 19136.8} C_VEL
LIN {X 0,Y 401.484,Z 290.222,A -85,B 0,C 180,E1 19132.838,E2 19132.838} C_VEL
LIN {X 0,Y 401.481,Z 290.223,A -85,B 0,C 180,E1 19128.894,E2 19128.894} C_VEL
LIN {X 0,Y 401.483,Z 290.223,A -85,B 0,C 180,E1 19124.988,E2 19124.988} C_VEL
LIN {X 0,Y 401.481,Z 290.224,A -85,B 0,C 180,E1 19121.012,E2 19121.012} C_VEL
LIN {X 0,Y 401.483,Z 290.223,A -85,B 0,C 180,E1 19117.062,E2 19117.062} C_VEL
LIN {X 0,Y 401.488,Z 290.222,A -85,B 0,C 180,E1 19113.202,E2 19113.202} C_VEL
LIN {X 0,Y 401.5,Z 290.22,A -85,B 0,C 180,E1 19109.357,E2 19109.357} C_VEL
LIN {X 0,Y 401.502,Z 290.224,A -85,B 0,C 180,E1 19105.52,E2 19105.52} C_VEL
LIN {X 0,Y 401.51,Z 290.222,A -85,B 0,C 180,E1 19101.627,E2 19101.627} C_VEL
LIN {X 0,Y 401.5,Z 290.216,A -85,B 0,C 180,E1 19097.687,E2 19097.687} C_VEL
LIN {X 0,Y 401.502,Z 290.21,A -85,B 0,C 180,E1 19093.685,E2 19093.685} C_VEL
LIN {X 0,Y 401.485,Z 290.184,A -85,B 0,C 180,E1 19089.75,E2 19089.75} C_VEL
LIN {X 0,Y 401.473,Z 290.225,A -85,B 0,C 180,E1 19086.004,E2 19086.004} C_VEL
LIN {X 0,Y 401.46,Z 290.199,A -85,B 0,C 180,E1 19082.141,E2 19082.141} C_VEL
LIN {X 0,Y 401.456,Z 290.196,A -85,B 0,C 180,E1 19078.287,E2 19078.287} C_VEL
LIN {X 0,Y 401.46,Z 290.228,A -85,B 0,C 180,E1 19074.283,E2 19074.283} C_VEL
LIN {X 0,Y 401.456,Z 290.191,A -85,B 0,C 180,E1 19070.394,E2 19070.394} C_VEL
LIN {X 0,Y 401.467,Z 290.206,A -85,B 0,C 180,E1 19066.608,E2 19066.608} C_VEL
LIN {X 0,Y 401.483,Z 290.221,A -85,B 0,C 180,E1 19062.761,E2 19062.761} C_VEL
LIN {X 0,Y 401.489,Z 290.19,A -85,B 0,C 180,E1 19058.832,E2 19058.832} C_VEL
LIN {X 0,Y 401.491,Z 290.194,A -85,B 0,C 180,E1 19054.953,E2 19054.953} C_VEL
LIN {X 0,Y 401.501,Z 290.21,A -85,B 0,C 180,E1 19050.935,E2 19050.935} C_VEL
LIN {X 0,Y 401.486,Z 290.21,A -85,B 0,C 180,E1 19046.948,E2 19046.948} C_VEL
LIN {X 0,Y 401.483,Z 290.49,A -85,B 0,C 180,E1 19045.748,E2 19045.748} C_VEL
LIN {X 0,Y 404.589,Z 298.092,A -85,B 0,C 180,E1 19043.534,E2 19043.534} C_VEL
LIN {X 0,Y 414.7,Z 313.033,A -85,B 0,C 180,E1 19041.269,E2 19041.269} C_VEL
LIN {X 0,Y 422.529,Z 324.887,A -85,B 0,C 180,E1 19039.669,E2 19039.669} C_VEL
LIN {X 0,Y 432.675,Z 341.555,A -85,B 0,C 180,E1 19037.72,E2 19037.72} C_VEL
LIN {X 0,Y 443.501,Z 360.901,A -85,B 0,C 180,E1 19035.775,E2 19035.775} C_VEL
LIN {X 0,Y 436.552,Z 571.278,A -85,B 0,C 180,E1 19031.988,E2 19031.988} C_VEL
LIN {X 0,Y 435.112,Z 608.92,A -85,B 0,C 180,E1 19031.271,E2 19031.271} C_VEL
LIN {X 0,Y 433.304,Z 630.619,A -85,B 0,C 180,E1 19030.641,E2 19030.641} C_VEL
LIN {X 0,Y 431.426,Z 648.725,A -85,B 0,C 180,E1 19029.937,E2 19029.937} C_VEL
LIN {X 0,Y 428.893,Z 669.5,A -85,B 0,C 180,E1 19028.912,E2 19028.912} C_VEL
LIN {X 0,Y 425.977,Z 688.972,A -85,B 0,C 180,E1 19027.693,E2 19027.693} C_VEL
LIN {X 0,Y 423.258,Z 705.649,A -85,B 0,C 180,E1 19026.448,E2 19026.448} C_VEL
LIN {X 0,Y 419.978,Z 724.592,A -85,B 0,C 180,E1 19024.78,E2 19024.78} C_VEL
LIN {X 0,Y 416.66,Z 742.065,A -85,B 0,C 180,E1 19022.923,E2 19022.923} C_VEL
LIN {X 0,Y 413.837,Z 756.649,A -85,B 0,C 180,E1 19021.133,E2 19021.133} C_VEL
LIN {X 0,Y 410.662,Z 773.169,A -85,B 0,C 180,E1 19018.776,E2 19018.776} C_VEL
LIN {X 0,Y 408.037,Z 786.759,A -85,B 0,C 180,E1 19016.485,E2 19016.485} C_VEL
LIN {X 0,Y 405.975,Z 798.136,A -85,B 0,C 180,E1 19014.286,E2 19014.286} C_VEL
LIN {X 0,Y 403.899,Z 810.608,A -85,B 0,C 180,E1 19011.492,E2 19011.492} C_VEL
LIN {X 0,Y 402.345,Z 820.955,A -85,B 0,C 180,E1 19008.697,E2 19008.697} C_VEL
LIN {X 0,Y 401.359,Z 828.821,A -85,B 0,C 180,E1 19006.201,E2 19006.201} C_VEL
LIN {X 0,Y 400.574,Z 836.841,A -85,B 0,C 180,E1 19003.128,E2 19003.128} C_VEL
LIN {X 0,Y 400.164,Z 842.672,A -85,B 0,C 180,E1 19000.218,E2 19000.218} C_VEL
LIN {X 0,Y 400.001,Z 846.481,A -85,B 0,C 180,E1 18997.757,E2 18997.757} C_VEL
LIN {X 0,Y 399.934,Z 849.371,A -85,B 0,C 180,E1 18995.164,E2 18995.164} C_VEL
LIN {X 0,Y 399.915,Z 851.359,A -85,B 0,C 180,E1 18992.006,E2 18992.006} C_VEL
LIN {X 0,Y 399.916,Z 851.58,A -85,B 0,C 180,E1 18989.14,E2 18989.14} C_VEL
LIN {X 0,Y 399.921,Z 850.708,A -85,B 0,C 180,E1 18986.704,E2 18986.704} C_VEL
LIN {X 0,Y 399.941,Z 848.82,A -85,B 0,C 180,E1 18984.261,E2 18984.261} C_VEL
LIN {X 0,Y 400.038,Z 845.51,A -85,B 0,C 180,E1 18981.52,E2 18981.52} C_VEL
LIN {X 0,Y 400.346,Z 839.753,A -85,B 0,C 180,E1 18978.241,E2 18978.241} C_VEL
LIN {X 0,Y 400.826,Z 833.954,A -85,B 0,C 180,E1 18975.703,E2 18975.703} C_VEL
LIN {X 0,Y 401.565,Z 827.089,A -85,B 0,C 180,E1 18973.213,E2 18973.213} C_VEL
LIN {X 0,Y 402.869,Z 817.421,A -85,B 0,C 180,E1 18970.274,E2 18970.274} C_VEL
LIN {X 0,Y 404.512,Z 806.659,A -85,B 0,C 180,E1 18967.584,E2 18967.584} C_VEL
LIN {X 0,Y 406.355,Z 795.978,A -85,B 0,C 180,E1 18965.274,E2 18965.274} C_VEL
LIN {X 0,Y 408.997,Z 781.872,A -85,B 0,C 180,E1 18962.64,E2 18962.64} C_VEL
LIN {X 0,Y 411.807,Z 767.043,A -85,B 0,C 180,E1 18960.311,E2 18960.311} C_VEL
LIN {X 0,Y 414.493,Z 753.326,A -85,B 0,C 180,E1 18958.437,E2 18958.437} C_VEL
LIN {X 0,Y 417.861,Z 735.864,A -85,B 0,C 180,E1 18956.376,E2 18956.376} C_VEL
LIN {X 0,Y 420.944,Z 718.941,A -85,B 0,C 180,E1 18954.7,E2 18954.7} C_VEL
LIN {X 0,Y 423.709,Z 703.04,A -85,B 0,C 180,E1 18953.344,E2 18953.344} C_VEL
LIN {X 0,Y 426.787,Z 684.035,A -85,B 0,C 180,E1 18951.966,E2 18951.966} C_VEL
LIN {X 0,Y 429.607,Z 663.651,A -85,B 0,C 180,E1 18950.78,E2 18950.78} C_VEL
LIN {X 0,Y 431.769,Z 645.591,A -85,B 0,C 180,E1 18949.928,E2 18949.928} C_VEL
LIN {X 0,Y 433.962,Z 624.031,A -85,B 0,C 180,E1 18949.137,E2 18949.137} C_VEL
LIN {X 0,Y 435.443,Z 602.282,A -85,B 0,C 180,E1 18948.591,E2 18948.591} C_VEL
LIN {X 0,Y 442.398,Z 393.667,A -85,B 0,C 180,E1 18944.82,E2 18944.82} C_VEL
LIN {X 0,Y 443.35,Z 360.627,A -85,B 0,C 180,E1 18944.199,E2 18944.199} C_VEL
LIN {X 0,Y 431.949,Z 340.273,A -85,B 0,C 180,E1 18942.143,E2 18942.143} C_VEL
LIN {X 0,Y 421.54,Z 323.325,A -85,B 0,C 180,E1 18940.133,E2 18940.133} C_VEL
LIN {X 0,Y 412.377,Z 309.559,A -85,B 0,C 180,E1 18938.235,E2 18938.235} C_VEL
LIN {X 0,Y 404.426,Z 297.698,A -85,B 0,C 180,E1 18936.395,E2 18936.395} C_VEL
LIN {X 0,Y 401.458,Z 290.327,A -85,B 0,C 180,E1 18934.156,E2 18934.156} C_VEL
LIN {X 0,Y 401.445,Z 290.208,A -85,B 0,C 180,E1 18930.205,E2 18930.205} C_VEL
LIN {X 0,Y 401.45,Z 290.197,A -85,B 0,C 180,E1 18926.316,E2 18926.316} C_VEL
LIN {X 0,Y 401.456,Z 290.216,A -85,B 0,C 180,E1 18922.399,E2 18922.399} C_VEL
LIN {X 0,Y 401.474,Z 290.213,A -85,B 0,C 180,E1 18918.589,E2 18918.589} C_VEL
LIN {X 0,Y 401.489,Z 290.184,A -85,B 0,C 180,E1 18914.715,E2 18914.715} C_VEL
LIN {X 0,Y 401.494,Z 290.206,A -85,B 0,C 180,E1 18910.765,E2 18910.765} C_VEL
LIN {X 0,Y 401.503,Z 290.215,A -85,B 0,C 180,E1 18906.721,E2 18906.721} C_VEL
LIN {X 0,Y 401.494,Z 290.182,A -85,B 0,C 180,E1 18902.712,E2 18902.712} C_VEL
LIN {X 0,Y 401.501,Z 290.215,A -85,B 0,C 180,E1 18898.858,E2 18898.858} C_VEL
LIN {X 0,Y 401.493,Z 290.205,A -85,B 0,C 180,E1 18894.856,E2 18894.856} C_VEL
LIN {X 0,Y 401.475,Z 290.189,A -85,B 0,C 180,E1 18891.118,E2 18891.118} C_VEL
LIN {X 0,Y 401.475,Z 290.228,A -85,B 0,C 180,E1 18887.194,E2 18887.194} C_VEL
LIN {X 0,Y 401.467,Z 290.198,A -85,B 0,C 180,E1 18883.357,E2 18883.357} C_VEL
LIN {X 0,Y 401.471,Z 290.225,A -85,B 0,C 180,E1 18879.442,E2 18879.442} C_VEL
LIN {X 0,Y 401.474,Z 290.227,A -85,B 0,C 180,E1 18875.424,E2 18875.424} C_VEL
LIN {X 0,Y 401.477,Z 290.227,A -85,B 0,C 180,E1 18871.434,E2 18871.434} C_VEL
LIN {X 0,Y 401.479,Z 290.227,A -85,B 0,C 180,E1 18867.457,E2 18867.457} C_VEL
LIN {X 0,Y 401.481,Z 290.227,A -85,B 0,C 180,E1 18863.472,E2 18863.472} C_VEL
LIN {X 0,Y 401.495,Z 290.225,A -85,B 0,C 180,E1 18859.643,E2 18859.643} C_VEL
LIN {X 0,Y 401.499,Z 290.224,A -85,B 0,C 180,E1 18855.79,E2 18855.79} C_VEL
LIN {X 0,Y 401.507,Z 290.223,A -85,B 0,C 180,E1 18851.865,E2 18851.865} C_VEL
LIN {X 0,Y 401.504,Z 290.225,A -85,B 0,C 180,E1 18847.869,E2 18847.869} C_VEL
LIN {X 0,Y 401.501,Z 290.225,A -85,B 0,C 180,E1 18843.905,E2 18843.905} C_VEL
LIN {X 0,Y 401.504,Z 290.222,A -85,B 0,C 180,E1 18839.871,E2 18839.871} C_VEL
LIN {X 0,Y 401.502,Z 290.22,A -85,B 0,C 180,E1 18835.836,E2 18835.836} C_VEL
LIN {X 0,Y 401.503,Z 290.22,A -85,B 0,C 180,E1 18831.934,E2 18831.934} C_VEL
LIN {X 0,Y 401.5,Z 290.219,A -85,B 0,C 180,E1 18827.956,E2 18827.956} C_VEL
LIN {X 0,Y 401.505,Z 290.219,A -85,B 0,C 180,E1 18823.978,E2 18823.978} C_VEL
LIN {X 0,Y 401.498,Z 290.22,A -85,B 0,C 180,E1 18820.039,E2 18820.039} C_VEL
LIN {X 0,Y 401.501,Z 290.22,A -85,B 0,C 180,E1 18816.147,E2 18816.147} C_VEL
LIN {X 0,Y 401.498,Z 290.223,A -85,B 0,C 180,E1 18812.141,E2 18812.141} C_VEL
LIN {X 0,Y 401.498,Z 290.224,A -85,B 0,C 180,E1 18808.288,E2 18808.288} C_VEL
LIN {X 0,Y 401.497,Z 290.225,A -85,B 0,C 180,E1 18804.283,E2 18804.283} C_VEL
LIN {X 0,Y 401.498,Z 290.223,A -85,B 0,C 180,E1 18800.395,E2 18800.395} C_VEL
LIN {X 0,Y 401.5,Z 290.221,A -85,B 0,C 180,E1 18796.462,E2 18796.462} C_VEL
LIN {X 0,Y 401.499,Z 290.221,A -85,B 0,C 180,E1 18792.718,E2 18792.718} C_VEL
LIN {X 0,Y 400.527,Z 290.344,A -85,B 0,C 180,E1 18791.619,E2 18791.619} C_VEL
LIN {X 0,Y 393.944,Z 291.162,A -85,B 0,C 180,E1 18788.359,E2 18788.359} C_VEL
LIN {X 0,Y 393.565,Z 291.211,A -85,B 0,C 180,E1 18787.71,E2 18787.71} C_VEL
LIN {X 0,Y 393.562,Z 291.214,A -85,B 0,C 180,E1 18783.741,E2 18783.741} C_VEL
LIN {X 0,Y 393.569,Z 291.212,A -85,B 0,C 180,E1 18779.742,E2 18779.742} C_VEL
LIN {X 0,Y 393.56,Z 291.21,A -85,B 0,C 180,E1 18775.657,E2 18775.657} C_VEL
LIN {X 0,Y 393.568,Z 291.209,A -85,B 0,C 180,E1 18771.694,E2 18771.694} C_VEL
LIN {X 0,Y 393.562,Z 291.209,A -85,B 0,C 180,E1 18767.671,E2 18767.671} C_VEL
LIN {X 0,Y 393.561,Z 291.208,A -85,B 0,C 180,E1 18763.611,E2 18763.611} C_VEL
LIN {X 0,Y 393.571,Z 291.207,A -85,B 0,C 180,E1 18759.617,E2 18759.617} C_VEL
LIN {X 0,Y 393.562,Z 291.208,A -85,B 0,C 180,E1 18755.576,E2 18755.576} C_VEL
LIN {X 0,Y 393.566,Z 291.208,A -85,B 0,C 180,E1 18751.557,E2 18751.557} C_VEL
LIN {X 0,Y 393.568,Z 291.212,A -85,B 0,C 180,E1 18747.54,E2 18747.54} C_VEL
LIN {X 0,Y 393.569,Z 291.213,A -85,B 0,C 180,E1 18743.496,E2 18743.496} C_VEL
LIN {X 0,Y 393.564,Z 291.213,A -85,B 0,C 180,E1 18739.439,E2 18739.439} C_VEL
LIN {X 0,Y 393.566,Z 291.171,A -85,B 0,C 180,E1 18735.471,E2 18735.471} C_VEL
LIN {X 0,Y 393.56,Z 291.195,A -85,B 0,C 180,E1 18731.43,E2 18731.43} C_VEL
LIN {X 0,Y 393.57,Z 291.202,A -85,B 0,C 180,E1 18727.444,E2 18727.444} C_VEL
LIN {X 0,Y 393.551,Z 291.17,A -85,B 0,C 180,E1 18723.496,E2 18723.496} C_VEL
LIN {X 0,Y 393.552,Z 291.206,A -85,B 0,C 180,E1 18719.563,E2 18719.563} C_VEL
LIN {X 0,Y 393.537,Z 291.19,A -85,B 0,C 180,E1 18715.629,E2 18715.629} C_VEL
LIN {X 0,Y 393.522,Z 291.179,A -85,B 0,C 180,E1 18711.82,E2 18711.82} C_VEL
LIN {X 0,Y 393.52,Z 291.217,A -85,B 0,C 180,E1 18707.975,E2 18707.975} C_VEL
LIN {X 0,Y 393.512,Z 291.185,A -85,B 0,C 180,E1 18704.073,E2 18704.073} C_VEL
LIN {X 0,Y 393.511,Z 291.183,A -85,B 0,C 180,E1 18700.067,E2 18700.067} C_VEL
LIN {X 0,Y 393.512,Z 291.207,A -85,B 0,C 180,E1 18696.013,E2 18696.013} C_VEL
LIN {X 0,Y 393.509,Z 291.219,A -85,B 0,C 180,E1 18691.962,E2 18691.962} C_VEL
LIN {X 0,Y 393.509,Z 291.221,A -85,B 0,C 180,E1 18687.924,E2 18687.924} C_VEL
LIN {X 0,Y 393.593,Z 291.561,A -85,B 0,C 180,E1 18687.069,E2 18687.069} C_VEL
LIN {X 0,Y 395.874,Z 297.422,A -85,B 0,C 180,E1 18685.282,E2 18685.282} C_VEL
LIN {X 0,Y 400.655,Z 303.972,A -85,B 0,C 180,E1 18684.094,E2 18684.094} C_VEL
LIN {X 0,Y 411.179,Z 319.564,A -85,B 0,C 180,E1 18681.7,E2 18681.7} C_VEL
LIN {X 0,Y 418.431,Z 330.652,A -85,B 0,C 180,E1 18680.179,E2 18680.179} C_VEL
LIN {X 0,Y 428.378,Z 347.209,A -85,B 0,C 180,E1 18678.212,E2 18678.212} C_VEL
LIN {X 0,Y 437.807,Z 364.301,A -85,B 0,C 180,E1 18676.461,E2 18676.461} C_VEL
LIN {X 0,Y 430.35,Z 579.071,A -85,B 0,C 180,E1 18672.558,E2 18672.558} C_VEL
LIN {X 0,Y 428.992,Z 610.078,A -85,B 0,C 180,E1 18671.943,E2 18671.943} C_VEL
LIN {X 0,Y 427.178,Z 630.786,A -85,B 0,C 180,E1 18671.33,E2 18671.33} C_VEL
LIN {X 0,Y 425.151,Z 649.424,A -85,B 0,C 180,E1 18670.595,E2 18670.595} C_VEL
LIN {X 0,Y 422.265,Z 671.417,A -85,B 0,C 180,E1 18669.474,E2 18669.474} C_VEL
LIN {X 0,Y 419.395,Z 689.708,A -85,B 0,C 180,E1 18668.304,E2 18668.304} C_VEL
LIN {X 0,Y 416.557,Z 706.265,A -85,B 0,C 180,E1 18667.046,E2 18667.046} C_VEL
LIN {X 0,Y 412.94,Z 725.863,A -85,B 0,C 180,E1 18665.273,E2 18665.273} C_VEL
LIN {X 0,Y 409.638,Z 742.426,A -85,B 0,C 180,E1 18663.478,E2 18663.478} C_VEL
LIN {X 0,Y 406.673,Z 756.946,A -85,B 0,C 180,E1 18661.662,E2 18661.662} C_VEL
LIN {X 0,Y 403.249,Z 773.682,A -85,B 0,C 180,E1 18659.216,E2 18659.216} C_VEL
LIN {X 0,Y 400.617,Z 786.57,A -85,B 0,C 180,E1 18657.001,E2 18657.001} C_VEL
LIN {X 0,Y 398.35,Z 798.316,A -85,B 0,C 180,E1 18654.685,E2 18654.685} C_VEL
LIN {X 0,Y 396.063,Z 811.152,A -85,B 0,C 180,E1 18651.719,E2 18651.719} C_VEL
LIN {X 0,Y 394.514,Z 820.859,A -85,B 0,C 180,E1 18649.033,E2 18649.033} C_VEL
LIN {X 0,Y 393.427,Z 828.999,A -85,B 0,C 180,E1 18646.385,E2 18646.385} C_VEL
LIN {X 0,Y 392.569,Z 837.208,A -85,B 0,C 180,E1 18643.101,E2 18643.101} C_VEL
LIN {X 0,Y 392.169,Z 842.671,A -85,B 0,C 180,E1 18640.28,E2 18640.28} C_VEL
LIN {X 0,Y 391.992,Z 846.618,A -85,B 0,C 180,E1 18637.622,E2 18637.622} C_VEL
LIN {X 0,Y 391.927,Z 849.793,A -85,B 0,C 180,E1 18634.536,E2 18634.536} C_VEL
LIN {X 0,Y 391.917,Z 851.221,A -85,B 0,C 180,E1 18631.462,E2 18631.462} C_VEL
LIN {X 0,Y 391.923,Z 851.304,A -85,B 0,C 180,E1 18628.977,E2 18628.977} C_VEL
LIN {X 0,Y 391.921,Z 850.377,A -85,B 0,C 180,E1 18626.49,E2 18626.49} C_VEL
LIN {X 0,Y 391.949,Z 848.294,A -85,B 0,C 180,E1 18623.85,E2 18623.85} C_VEL
LIN {X 0,Y 392.097,Z 844.179,A -85,B 0,C 180,E1 18620.607,E2 18620.607} C_VEL
LIN {X 0,Y 392.414,Z 839.068,A -85,B 0,C 180,E1 18617.791,E2 18617.791} C_VEL
LIN {X 0,Y 392.947,Z 833.231,A -85,B 0,C 180,E1 18615.22,E2 18615.22} C_VEL
LIN {X 0,Y 393.875,Z 825.533,A -85,B 0,C 180,E1 18612.418,E2 18612.418} C_VEL
LIN {X 0,Y 395.404,Z 815.115,A -85,B 0,C 180,E1 18609.328,E2 18609.328} C_VEL
LIN {X 0,Y 397.061,Z 805.299,A -85,B 0,C 180,E1 18606.87,E2 18606.87} C_VEL
LIN {X 0,Y 399.418,Z 792.844,A -85,B 0,C 180,E1 18604.179,E2 18604.179} C_VEL
LIN {X 0,Y 402.155,Z 778.928,A -85,B 0,C 180,E1 18601.65,E2 18601.65} C_VEL
LIN {X 0,Y 404.849,Z 765.79,A -85,B 0,C 180,E1 18599.584,E2 18599.584} C_VEL
LIN {X 0,Y 408.108,Z 750.081,A -85,B 0,C 180,E1 18597.436,E2 18597.436} C_VEL
LIN {X 0,Y 411.706,Z 732.062,A -85,B 0,C 180,E1 18595.37,E2 18595.37} C_VEL
LIN {X 0,Y 414.582,Z 717.053,A -85,B 0,C 180,E1 18593.894,E2 18593.894} C_VEL
LIN {X 0,Y 417.659,Z 700.178,A -85,B 0,C 180,E1 18592.465,E2 18592.465} C_VEL
LIN {X 0,Y 421.044,Z 679.327,A -85,B 0,C 180,E1 18591.003,E2 18591.003} C_VEL
LIN {X 0,Y 423.643,Z 661.251,A -85,B 0,C 180,E1 18589.975,E2 18589.975} C_VEL
LIN {X 0,Y 426.03,Z 642.023,A -85,B 0,C 180,E1 18589.087,E2 18589.087} C_VEL
LIN {X 0,Y 428.257,Z 619.361,A -85,B 0,C 180,E1 18588.311,E2 18588.311} C_VEL
LIN {X 0,Y 429.536,Z 600.364,A -85,B 0,C 180,E1 18587.848,E2 18587.848} C_VEL
LIN {X 0,Y 437.049,Z 385.538,A -85,B 0,C 180,E1 18583.928,E2 18583.928} C_VEL
LIN {X 0,Y 437.667,Z 363.939,A -85,B 0,C 180,E1 18583.511,E2 18583.511} C_VEL
LIN {X 0,Y 427.298,Z 345.329,A -85,B 0,C 180,E1 18581.58,E2 18581.58} C_VEL
LIN {X 0,Y 417.593,Z 329.328,A -85,B 0,C 180,E1 18579.649,E2 18579.649} C_VEL
LIN {X 0,Y 408.82,Z 315.947,A -85,B 0,C 180,E1 18577.781,E2 18577.781} C_VEL
LIN {X 0,Y 399.991,Z 303.26,A -85,B 0,C 180,E1 18575.754,E2 18575.754} C_VEL
LIN {X 0,Y 395.589,Z 296.878,A -85,B 0,C 180,E1 18574.593,E2 18574.593} C_VEL
LIN {X 0,Y 393.542,Z 291.295,A -85,B 0,C 180,E1 18572.806,E2 18572.806} C_VEL
LIN {X 0,Y 393.545,Z 291.204,A -85,B 0,C 180,E1 18568.863,E2 18568.863} C_VEL
LIN {X 0,Y 393.546,Z 291.183,A -85,B 0,C 180,E1 18564.908,E2 18564.908} C_VEL
LIN {X 0,Y 393.555,Z 291.173,A -85,B 0,C 180,E1 18560.991,E2 18560.991} C_VEL
LIN {X 0,Y 393.557,Z 291.2,A -85,B 0,C 180,E1 18556.988,E2 18556.988} C_VEL
LIN {X 0,Y 393.553,Z 291.196,A -85,B 0,C 180,E1 18553.068,E2 18553.068} C_VEL
LIN {X 0,Y 393.547,Z 291.171,A -85,B 0,C 180,E1 18549.063,E2 18549.063} C_VEL
LIN {X 0,Y 393.541,Z 291.208,A -85,B 0,C 180,E1 18545.18,E2 18545.18} C_VEL
LIN {X 0,Y 393.54,Z 291.191,A -85,B 0,C 180,E1 18541.165,E2 18541.165} C_VEL
LIN {X 0,Y 393.525,Z 291.178,A -85,B 0,C 180,E1 18537.379,E2 18537.379} C_VEL
LIN {X 0,Y 393.529,Z 291.217,A -85,B 0,C 180,E1 18533.416,E2 18533.416} C_VEL
LIN {X 0,Y 393.524,Z 291.181,A -85,B 0,C 180,E1 18529.459,E2 18529.459} C_VEL
LIN {X 0,Y 393.525,Z 291.184,A -85,B 0,C 180,E1 18525.468,E2 18525.468} C_VEL
LIN {X 0,Y 393.533,Z 291.216,A -85,B 0,C 180,E1 18521.483,E2 18521.483} C_VEL
LIN {X 0,Y 393.533,Z 291.216,A -85,B 0,C 180,E1 18517.44,E2 18517.44} C_VEL
LIN {X 0,Y 393.536,Z 291.214,A -85,B 0,C 180,E1 18513.419,E2 18513.419} C_VEL
LIN {X 0,Y 393.539,Z 291.216,A -85,B 0,C 180,E1 18509.459,E2 18509.459} C_VEL
LIN {X 0,Y 393.542,Z 291.216,A -85,B 0,C 180,E1 18505.489,E2 18505.489} C_VEL
LIN {X 0,Y 393.545,Z 291.215,A -85,B 0,C 180,E1 18501.49,E2 18501.49} C_VEL
LIN {X 0,Y 393.556,Z 291.214,A -85,B 0,C 180,E1 18497.671,E2 18497.671} C_VEL
LIN {X 0,Y 393.557,Z 291.214,A -85,B 0,C 180,E1 18493.609,E2 18493.609} C_VEL
LIN {X 0,Y 393.562,Z 291.213,A -85,B 0,C 180,E1 18489.617,E2 18489.617} C_VEL
LIN {X 0,Y 393.559,Z 291.212,A -85,B 0,C 180,E1 18485.575,E2 18485.575} C_VEL
LIN {X 0,Y 393.564,Z 291.209,A -85,B 0,C 180,E1 18481.556,E2 18481.556} C_VEL
LIN {X 0,Y 393.564,Z 291.208,A -85,B 0,C 180,E1 18477.54,E2 18477.54} C_VEL
LIN {X 0,Y 393.566,Z 291.207,A -85,B 0,C 180,E1 18473.491,E2 18473.491} C_VEL
LIN {X 0,Y 393.584,Z 291.369,A -85,B 0,C 180,E1 18469.438,E2 18469.438} C_VEL
LIN {X 0,Y 393.953,Z 292.87,A -85,B 0,C 180,E1 18465.866,E2 18465.866} C_VEL
LIN {X 0,Y 394.794,Z 294.598,A -85,B 0,C 180,E1 18462.728,E2 18462.728} C_VEL
LIN {X 0,Y 395.594,Z 295.619,A -85,B 0,C 180,E1 18459.309,E2 18459.309} C_VEL
LIN {X 0,Y 396.174,Z 296.198,A -85,B 0,C 180,E1 18455.648,E2 18455.648} C_VEL
LIN {X 0,Y 396.465,Z 296.442,A -85,B 0,C 180,E1 18452.023,E2 18452.023} C_VEL
LIN {X 0,Y 396.464,Z 296.44,A -85,B 0,C 180,E1 18448.555,E2 18448.555} C_VEL
LIN {X 0,Y 396.213,Z 296.226,A -85,B 0,C 180,E1 18445.078,E2 18445.078} C_VEL
LIN {X 0,Y 395.707,Z 295.743,A -85,B 0,C 180,E1 18441.573,E2 18441.573} C_VEL
LIN {X 0,Y 394.962,Z 294.831,A -85,B 0,C 180,E1 18438.019,E2 18438.019} C_VEL
LIN {X 0,Y 394.161,Z 293.406,A -85,B 0,C 180,E1 18434.855,E2 18434.855} C_VEL
LIN {X 0,Y 393.612,Z 291.609,A -85,B 0,C 180,E1 18431.351,E2 18431.351} C_VEL
LIN {X 0,Y 393.565,Z 291.211,A -85,B 0,C 180,E1 18427.71,E2 18427.71} C_VEL
LIN {X 0,Y 392.902,Z 292.02,A -85,B 0,C 180,E1 18426.589,E2 18426.589} C_VEL
LIN {X 0,Y 389.022,Z 296.25,A -85,B 0,C 180,E1 18423.928,E2 18423.928} C_VEL
LIN {X 0,Y 387.822,Z 296.755,A -85,B 0,C 180,E1 18422.797,E2 18422.797} C_VEL
LIN {X 0,Y 387.725,Z 296.681,A -85,B 0,C 180,E1 18422.634,E2 18422.634} C_VEL
LIN {X 0,Y 386.201,Z 294.327,A -85,B 0,C 180,E1 18419.766,E2 18419.766} C_VEL
LIN {X 0,Y 385.689,Z 292.625,A -85,B 0,C 180,E1 18417.898,E2 18417.898} C_VEL
LIN {X 0,Y 385.613,Z 292.199,A -85,B 0,C 180,E1 18414.676,E2 18414.676} C_VEL
LIN {X 0,Y 385.613,Z 292.201,A -85,B 0,C 180,E1 18410.595,E2 18410.595} C_VEL
LIN {X 0,Y 385.611,Z 292.202,A -85,B 0,C 180,E1 18406.599,E2 18406.599} C_VEL
LIN {X 0,Y 385.609,Z 292.204,A -85,B 0,C 180,E1 18402.577,E2 18402.577} C_VEL
LIN {X 0,Y 385.602,Z 292.204,A -85,B 0,C 180,E1 18398.675,E2 18398.675} C_VEL
LIN {X 0,Y 385.602,Z 292.205,A -85,B 0,C 180,E1 18394.601,E2 18394.601} C_VEL
LIN {X 0,Y 385.6,Z 292.205,A -85,B 0,C 180,E1 18390.546,E2 18390.546} C_VEL
LIN {X 0,Y 385.599,Z 292.203,A -85,B 0,C 180,E1 18386.487,E2 18386.487} C_VEL
LIN {X 0,Y 385.594,Z 292.205,A -85,B 0,C 180,E1 18382.567,E2 18382.567} C_VEL
LIN {X 0,Y 385.594,Z 292.206,A -85,B 0,C 180,E1 18378.599,E2 18378.599} C_VEL
LIN {X 0,Y 385.586,Z 292.17,A -85,B 0,C 180,E1 18374.568,E2 18374.568} C_VEL
LIN {X 0,Y 385.587,Z 292.169,A -85,B 0,C 180,E1 18370.609,E2 18370.609} C_VEL
LIN {X 0,Y 385.589,Z 292.206,A -85,B 0,C 180,E1 18366.551,E2 18366.551} C_VEL
LIN {X 0,Y 385.584,Z 292.166,A -85,B 0,C 180,E1 18362.527,E2 18362.527} C_VEL
LIN {X 0,Y 385.59,Z 292.176,A -85,B 0,C 180,E1 18358.663,E2 18358.663} C_VEL
LIN {X 0,Y 385.593,Z 292.2,A -85,B 0,C 180,E1 18354.644,E2 18354.644} C_VEL
LIN {X 0,Y 385.596,Z 292.161,A -85,B 0,C 180,E1 18350.749,E2 18350.749} C_VEL
LIN {X 0,Y 385.604,Z 292.183,A -85,B 0,C 180,E1 18346.81,E2 18346.81} C_VEL
LIN {X 0,Y 385.616,Z 292.192,A -85,B 0,C 180,E1 18342.963,E2 18342.963} C_VEL
LIN {X 0,Y 385.612,Z 292.165,A -85,B 0,C 180,E1 18338.874,E2 18338.874} C_VEL
LIN {X 0,Y 385.61,Z 292.17,A -85,B 0,C 180,E1 18334.998,E2 18334.998} C_VEL
LIN {X 0,Y 385.622,Z 292.186,A -85,B 0,C 180,E1 18330.899,E2 18330.899} C_VEL
LIN {X 0,Y 385.636,Z 292.46,A -85,B 0,C 180,E1 18328.552,E2 18328.552} C_VEL
LIN {X 0,Y 387.504,Z 296.944,A -85,B 0,C 180,E1 18327.102,E2 18327.102} C_VEL
LIN {X 0,Y 392.191,Z 303.487,A -85,B 0,C 180,E1 18325.84,E2 18325.84} C_VEL
LIN {X 0,Y 398.745,Z 312.814,A -85,B 0,C 180,E1 18324.206,E2 18324.206} C_VEL
LIN {X 0,Y 407.08,Z 325.116,A -85,B 0,C 180,E1 18322.275,E2 18322.275} C_VEL
LIN {X 0,Y 414.571,Z 336.773,A -85,B 0,C 180,E1 18320.654,E2 18320.654} C_VEL
LIN {X 0,Y 424.184,Z 352.993,A -85,B 0,C 180,E1 18318.7,E2 18318.7} C_VEL
LIN {X 0,Y 432.172,Z 367.64,A -85,B 0,C 180,E1 18317.168,E2 18317.168} C_VEL
LIN {X 0,Y 424.317,Z 583.146,A -85,B 0,C 180,E1 18313.212,E2 18313.212} C_VEL
LIN {X 0,Y 422.901,Z 611.504,A -85,B 0,C 180,E1 18312.625,E2 18312.625} C_VEL
LIN {X 0,Y 421.087,Z 631.245,A -85,B 0,C 180,E1 18312.029,E2 18312.029} C_VEL
LIN {X 0,Y 418.954,Z 649.947,A -85,B 0,C 180,E1 18311.28,E2 18311.28} C_VEL
LIN {X 0,Y 415.85,Z 672.275,A -85,B 0,C 180,E1 18310.117,E2 18310.117} C_VEL
LIN {X 0,Y 413.034,Z 689.455,A -85,B 0,C 180,E1 18309.005,E2 18309.005} C_VEL
LIN {X 0,Y 410.064,Z 706.011,A -85,B 0,C 180,E1 18307.734,E2 18307.734} C_VEL
LIN {X 0,Y 406.402,Z 724.92,A -85,B 0,C 180,E1 18306.014,E2 18306.014} C_VEL
LIN {X 0,Y 402.916,Z 741.553,A -85,B 0,C 180,E1 18304.198,E2 18304.198} C_VEL
LIN {X 0,Y 399.781,Z 756.136,A -85,B 0,C 180,E1 18302.358,E2 18302.358} C_VEL
LIN {X 0,Y 396.262,Z 772.406,A -85,B 0,C 180,E1 18299.972,E2 18299.972} C_VEL
LIN {X 0,Y 393.262,Z 786.244,A -85,B 0,C 180,E1 18297.563,E2 18297.563} C_VEL
LIN {X 0,Y 390.911,Z 797.62,A -85,B 0,C 180,E1 18295.286,E2 18295.286} C_VEL
LIN {X 0,Y 388.538,Z 810.094,A -85,B 0,C 180,E1 18292.386,E2 18292.386} C_VEL
LIN {X 0,Y 386.749,Z 820.443,A -85,B 0,C 180,E1 18289.481,E2 18289.481} C_VEL
LIN {X 0,Y 385.61,Z 828.311,A -85,B 0,C 180,E1 18286.882,E2 18286.882} C_VEL
LIN {X 0,Y 384.685,Z 836.333,A -85,B 0,C 180,E1 18283.681,E2 18283.681} C_VEL
LIN {X 0,Y 384.211,Z 842.168,A -85,B 0,C 180,E1 18280.647,E2 18280.647} C_VEL
LIN {X 0,Y 384.021,Z 845.98,A -85,B 0,C 180,E1 18278.082,E2 18278.082} C_VEL
LIN {X 0,Y 383.94,Z 848.872,A -85,B 0,C 180,E1 18275.379,E2 18275.379} C_VEL
LIN {X 0,Y 383.923,Z 850.862,A -85,B 0,C 180,E1 18272.089,E2 18272.089} C_VEL
LIN {X 0,Y 383.924,Z 851.083,A -85,B 0,C 180,E1 18269.105,E2 18269.105} C_VEL
LIN {X 0,Y 383.924,Z 850.211,A -85,B 0,C 180,E1 18266.566,E2 18266.566} C_VEL
LIN {X 0,Y 383.948,Z 848.321,A -85,B 0,C 180,E1 18264.021,E2 18264.021} C_VEL
LIN {X 0,Y 384.042,Z 845.202,A -85,B 0,C 180,E1 18261.315,E2 18261.315} C_VEL
LIN {X 0,Y 384.388,Z 839.704,A -85,B 0,C 180,E1 18257.97,E2 18257.97} C_VEL
LIN {X 0,Y 384.98,Z 833.445,A -85,B 0,C 180,E1 18255.101,E2 18255.101} C_VEL
LIN {X 0,Y 385.857,Z 826.485,A -85,B 0,C 180,E1 18252.474,E2 18252.474} C_VEL
LIN {X 0,Y 387.441,Z 816.34,A -85,B 0,C 180,E1 18249.296,E2 18249.296} C_VEL
LIN {X 0,Y 389.332,Z 805.683,A -85,B 0,C 180,E1 18246.544,E2 18246.544} C_VEL
LIN {X 0,Y 391.498,Z 794.744,A -85,B 0,C 180,E1 18244.106,E2 18244.106} C_VEL
LIN {X 0,Y 394.701,Z 779.518,A -85,B 0,C 180,E1 18241.221,E2 18241.221} C_VEL
LIN {X 0,Y 397.516,Z 766.529,A -85,B 0,C 180,E1 18239.129,E2 18239.129} C_VEL
LIN {X 0,Y 400.502,Z 752.813,A -85,B 0,C 180,E1 18237.199,E2 18237.199} C_VEL
LIN {X 0,Y 404.237,Z 735.448,A -85,B 0,C 180,E1 18235.094,E2 18235.094} C_VEL
LIN {X 0,Y 407.729,Z 718.106,A -85,B 0,C 180,E1 18233.337,E2 18233.337} C_VEL
LIN {X 0,Y 410.717,Z 702.533,A -85,B 0,C 180,E1 18231.983,E2 18231.983} C_VEL
LIN {X 0,Y 414.08,Z 683.529,A -85,B 0,C 180,E1 18230.577,E2 18230.577} C_VEL
LIN {X 0,Y 417.155,Z 663.28,A -85,B 0,C 180,E1 18229.379,E2 18229.379} C_VEL
LIN {X 0,Y 419.54,Z 645.09,A -85,B 0,C 180,E1 18228.508,E2 18228.508} C_VEL
LIN {X 0,Y 421.929,Z 623.531,A -85,B 0,C 180,E1 18227.708,E2 18227.708} C_VEL
LIN {X 0,Y 423.526,Z 601.783,A -85,B 0,C 180,E1 18227.153,E2 18227.153} C_VEL
LIN {X 0,Y 431.209,Z 393.278,A -85,B 0,C 180,E1 18223.306,E2 18223.306} C_VEL
LIN {X 0,Y 432.089,Z 367.276,A -85,B 0,C 180,E1 18222.812,E2 18222.812} C_VEL
LIN {X 0,Y 420.861,Z 347.105,A -85,B 0,C 180,E1 18220.636,E2 18220.636} C_VEL
LIN {X 0,Y 409.45,Z 328.622,A -85,B 0,C 180,E1 18218.246,E2 18218.246} C_VEL
LIN {X 0,Y 399.647,Z 314.118,A -85,B 0,C 180,E1 18216.011,E2 18216.011} C_VEL
LIN {X 0,Y 396.316,Z 309.381,A -85,B 0,C 180,E1 18215.203,E2 18215.203} C_VEL
LIN {X 0,Y 389.834,Z 300.508,A -85,B 0,C 180,E1 18213.554,E2 18213.554} C_VEL
LIN {X 0,Y 387.229,Z 296.25,A -85,B 0,C 180,E1 18212.748,E2 18212.748} C_VEL
LIN {X 0,Y 385.625,Z 292.37,A -85,B 0,C 180,E1 18211.41,E2 18211.41} C_VEL
LIN {X 0,Y 385.592,Z 292.189,A -85,B 0,C 180,E1 18207.488,E2 18207.488} C_VEL
